   // sequencer 2: S100-S199 等待到位 / S100-S199 CheckLineMode
   STEP ProcessStart:   // S100, max time T#10S, warning time T#7S
      // 自动等待开始运行
              R    #ioPM_Inface.InitialRun
              R    #ioPM_Inface.ProcessComplete
              R    #ioPM_Inface.ProcessStart
              S    #ioPM_Inface.InitialOK
              S    #ioPM_Inface.WaitRunning
          S1  N    #ioPM_Inface.ProcessResult:=0
   END_STEP
   TRANSITION Trans200 FROM ProcessStart TO MotorRun   // T100
      := TRUE;
   END_TRANSITION
   STEP "Process Finish_1":   // S237, max time T#10S, warning time T#7S
   END_STEP
   TRANSITION Trans250 FROM "Process Finish_1" TO "CheckMachine Mode_1"   // T249, jump
      := TRUE;
   END_TRANSITION
   STEP StopProcess:   // S27, max time T#10S, warning time T#7S
   END_STEP
   TRANSITION Trans34 FROM StopProcess TO (UnloadStoper_1, UnloadStoper_2, UnloadStoper_3, "CheckMachine Mode_1", "CheckMachine Mode_2", "CheckMachine Mode_3", "CheckMachine Mode_4")   // T33
      := TRUE;
   END_TRANSITION
   STEP MotorRun:   // S34, max time T#10S, warning time T#7S
              S    "MotorControl".Dev[11].Auto.Start
              R    "MotorControl".Dev[11].Auto.CCWStart
              S    "MotorControl".Dev[12].Auto.Start
              R    "MotorControl".Dev[12].Auto.CCWStart
   END_STEP
   TRANSITION Trans39 FROM MotorRun TO StopProcess   // T38
      := TRUE;
   END_TRANSITION
   STEP LoadingStop_4:   // S30, max time T#10S, warning time T#7S
   END_STEP
   TRANSITION Trans122 FROM LoadingStop_4 TO CheckPalletExist_3   // T122
      := TRUE;
   END_TRANSITION
   STEP LoadingStop_2:   // S28, max time T#10S, warning time T#7S
   END_STEP
   TRANSITION Trans120 FROM LoadingStop_2 TO CheckPalletExist_1   // T120
      := TRUE;
   END_TRANSITION
   STEP "CheckMachine Mode_3":   // S156, max time T#10S, warning time T#7S
   END_STEP
   TRANSITION Trans166 FROM "CheckMachine Mode_3" TO LoadingStop_3   // T166
      := NOT "AutoProcessControl".Global.H.EmptyPallet;
   END_TRANSITION
   STEP LoadingStop_3:   // S29, max time T#10S, warning time T#7S
   END_STEP
   TRANSITION Trans121 FROM LoadingStop_3 TO CheckPalletExist_2   // T121
      := TRUE;
   END_TRANSITION
   STEP CheckPalletExist:   // S31, max time T#10S, warning time T#7S
              R    "MotorControl".Dev[11].Auto.CCWStart
   END_STEP
   TRANSITION Trans35 FROM CheckPalletExist TO WaitLineMotorReady   // T34
      := "iH-shaftLoadingDetection1" AND (#CheckPalletExist.T > t#1000MS) AND NOT "AutoProcessControl".Robot_1.ClearPart;
   END_TRANSITION
   STEP AriveTimeDelay_1:   // S119, max time T#10S, warning time T#7S
   END_STEP
   TRANSITION Trans119 FROM AriveTimeDelay_1 TO StoperReset_1   // T119
      := #AriveTimeDelay_1.T > t#500MS;
   END_TRANSITION
   STEP WaitLineMotorReady:   // S35, max time T#10S, warning time T#7S
   END_STEP
   TRANSITION Trans40 FROM WaitLineMotorReady TO WaitPalletRequestRelease   // T39
      := "MotorControl".Dev[11].OutControl.o_Ready;
   END_TRANSITION
   STEP WaitPalletRequestRelease:   // S36, max time T#10S, warning time T#7S
   END_STEP
   TRANSITION Trans41 FROM WaitPalletRequestRelease TO StoperRelease_1   // T40
      := "AutoProcessControl".Global.H.LoadStopRequestPallet_1;
   END_TRANSITION
   TRANSITION Trans207 FROM WaitPalletRequestRelease TO "CheckMachine Mode_1"   // T207, jump
      := "AutoProcessControl".Global.H.EmptyPallet;
   END_TRANSITION
   STEP LoadingStop_1:   // S142, max time T#10S, warning time T#7S
   END_STEP
   TRANSITION Trans776 FROM LoadingStop_1 TO CheckPalletExist   // T141
      := TRUE;
   END_TRANSITION
   STEP WaitPalletArrveNextPos:   // S37, max time T#10S, warning time T#7S
              S    "MotorControl".Dev[11].Auto.Start
              R    "MotorControl".Dev[11].Auto.CCWStart
   END_STEP
   TRANSITION Trans42 FROM WaitPalletArrveNextPos TO AriveTimeDelay_1   // T41
      := "iH-shaftLoadingDetection2" OR "AutoProcessControl".Global.H.EmptyPallet;
   END_TRANSITION
   STEP "Process Finish_2":   // S238, max time T#10S, warning time T#7S
   END_STEP
   TRANSITION Trans251 FROM "Process Finish_2" TO "CheckMachine Mode_2"   // T250, jump
      := TRUE;
   END_TRANSITION
   STEP StoperReset_1:   // S117, max time T#10S, warning time T#7S
              S    "ST10Cylinder".Cy[23].Inout.AutoGoHome
              R    "ST10Cylinder".Cy[23].Inout.AutoGoWork
   END_STEP
   TRANSITION Trans766 FROM StoperReset_1 TO "Process Finish_1"   // T117
      := TRUE;
   END_TRANSITION
   STEP StoperRelease_1:   // S118, max time T#10S, warning time T#7S
              R    "ST10Cylinder".Cy[23].Inout.AutoGoHome
              S    "ST10Cylinder".Cy[23].Inout.AutoGoWork
   END_STEP
   TRANSITION Trans767 FROM StoperRelease_1 TO WaitPalletArrveNextPos   // T118
      := #StoperRelease_1.T > t#1000MS;
   END_TRANSITION
   STEP CheckPalletExist_1:   // S32, max time T#10S, warning time T#7S
   END_STEP
   TRANSITION Trans36 FROM CheckPalletExist_1 TO WaitLineMotorReady_1   // T35
      := "iH-shaftLoadingDetection2" AND (#CheckPalletExist_1.T > t#1000MS);
   END_TRANSITION
   TRANSITION Trans126 FROM CheckPalletExist_1 TO WaitPalletArive   // T126
      := NOT "iH-shaftLoadingDetection2" AND (#CheckPalletExist_1.T > t#1000MS);
   END_TRANSITION
   STEP AriveTimeDelay_2:   // S120, max time T#10S, warning time T#7S
   END_STEP
   TRANSITION Trans123 FROM AriveTimeDelay_2 TO StoperReset_2   // T123
      := #AriveTimeDelay_2.T > t#500MS;
   END_TRANSITION
   STEP WaitLineMotorReady_1:   // S38, max time T#10S, warning time T#7S
   END_STEP
   TRANSITION Trans44 FROM WaitLineMotorReady_1 TO WaitPalletRequestRelease_1   // T43
      := "MotorControl".Dev[11].OutControl.o_Ready;
   END_TRANSITION
   STEP WaitPalletRequestRelease_1:   // S39, max time T#10S, warning time T#7S
   END_STEP
   TRANSITION Trans45 FROM WaitPalletRequestRelease_1 TO StoperRelease_2   // T44
      := "AutoProcessControl".Global.H.LoadStopRequestPallet_2;
   END_TRANSITION
   TRANSITION Trans206 FROM WaitPalletRequestRelease_1 TO "CheckMachine Mode_2"   // T206, jump
      := "AutoProcessControl".Global.H.EmptyPallet;
   END_TRANSITION
   STEP WaitPalletArrveNextPos_1:   // S40, max time T#10S, warning time T#7S
              S    "MotorControl".Dev[11].Auto.Start
              R    "MotorControl".Dev[11].Auto.CCWStart
   END_STEP
   TRANSITION Trans43 FROM WaitPalletArrveNextPos_1 TO AriveTimeDelay_2   // T42
      := "iH-shaftLoadingDetection3" OR "AutoProcessControl".Global.H.EmptyPallet;
   END_TRANSITION
   STEP StoperReset_2:   // S121, max time T#10S, warning time T#7S
              S    "ST10Cylinder".Cy[24].Inout.AutoGoHome
              R    "ST10Cylinder".Cy[24].Inout.AutoGoWork
   END_STEP
   TRANSITION Trans768 FROM StoperReset_2 TO "Process Finish_2"   // T124
      := TRUE;
   END_TRANSITION
   STEP StoperRelease_2:   // S122, max time T#10S, warning time T#7S
              R    "ST10Cylinder".Cy[24].Inout.AutoGoHome
              S    "ST10Cylinder".Cy[24].Inout.AutoGoWork
   END_STEP
   TRANSITION Trans769 FROM StoperRelease_2 TO WaitPalletArrveNextPos_1   // T125
      := #StoperRelease_2.T > t#1000MS;
   END_TRANSITION
   STEP WaitPalletArive:   // S123, max time T#10S, warning time T#7S
              N    "AutoProcessControl".Global.H.LoadStopRequestPallet_1
   END_STEP
   TRANSITION Trans127 FROM WaitPalletArive TO TimeDelay   // T127
      := "iH-shaftLoadingDetection2" OR "AutoProcessControl".Global.H.EmptyPallet;
   END_TRANSITION
   STEP TimeDelay:   // S124, max time T#10S, warning time T#7S
   END_STEP
   TRANSITION Trans128 FROM TimeDelay TO "CheckMachine Mode_2"   // T128, jump
      := #TimeDelay.T > t#500MS;
   END_TRANSITION
   STEP "Process Finish_3":   // S239, max time T#10S, warning time T#7S
   END_STEP
   TRANSITION Trans252 FROM "Process Finish_3" TO "CheckMachine Mode_3"   // T251, jump
      := TRUE;
   END_TRANSITION
   STEP CheckPalletExist_2:   // S41, max time T#10S, warning time T#7S
   END_STEP
   TRANSITION Trans37 FROM CheckPalletExist_2 TO WaitLineMotorReady_2   // T36
      := "iH-shaftLoadingDetection3" AND (#CheckPalletExist_2.T > t#1000MS);
   END_TRANSITION
   TRANSITION Trans129 FROM CheckPalletExist_2 TO WaitPalletArive_1   // T132
      := NOT "iH-shaftLoadingDetection3" AND (#CheckPalletExist_2.T > t#1000MS);
   END_TRANSITION
   STEP AriveTimeDelay_3:   // S125, max time T#10S, warning time T#7S
   END_STEP
   TRANSITION Trans124 FROM AriveTimeDelay_3 TO StoperReset_3   // T129
      := #AriveTimeDelay_3.T > t#500MS;
   END_TRANSITION
   STEP WaitLineMotorReady_2:   // S42, max time T#10S, warning time T#7S
   END_STEP
   TRANSITION Trans47 FROM WaitLineMotorReady_2 TO WaitPalletRequestRelease_2   // T46
      := "MotorControl".Dev[11].OutControl.o_Ready;
   END_TRANSITION
   STEP WaitPalletRequestRelease_2:   // S43, max time T#10S, warning time T#7S
   END_STEP
   TRANSITION Trans48 FROM WaitPalletRequestRelease_2 TO StoperRelease_3   // T47
      := "AutoProcessControl".Global.H.LoadStopRequestPallet_3;
   END_TRANSITION
   TRANSITION Trans205 FROM WaitPalletRequestRelease_2 TO "CheckMachine Mode_3"   // T205, jump
      := "AutoProcessControl".Global.H.EmptyPallet;
   END_TRANSITION
   STEP WaitPalletArrveNextPos_2:   // S44, max time T#10S, warning time T#7S
              S    "MotorControl".Dev[11].Auto.Start
              R    "MotorControl".Dev[11].Auto.CCWStart
   END_STEP
   TRANSITION Trans46 FROM WaitPalletArrveNextPos_2 TO AriveTimeDelay_3   // T45
      := "iH-shaftLoadingDetection4" OR "AutoProcessControl".Global.H.EmptyPallet;
   END_TRANSITION
   STEP StoperReset_3:   // S126, max time T#10S, warning time T#7S
              S    "ST10Cylinder".Cy[25].Inout.AutoGoHome
              R    "ST10Cylinder".Cy[25].Inout.AutoGoWork
   END_STEP
   TRANSITION Trans770 FROM StoperReset_3 TO "Process Finish_3"   // T130
      := TRUE;
   END_TRANSITION
   STEP StoperRelease_3:   // S127, max time T#10S, warning time T#7S
              R    "ST10Cylinder".Cy[25].Inout.AutoGoHome
              S    "ST10Cylinder".Cy[25].Inout.AutoGoWork
   END_STEP
   TRANSITION Trans771 FROM StoperRelease_3 TO WaitPalletArrveNextPos_2   // T131
      := #StoperRelease_3.T > t#1000MS;
   END_TRANSITION
   STEP WaitPalletArive_1:   // S128, max time T#10S, warning time T#7S
              N    "AutoProcessControl".Global.H.LoadStopRequestPallet_2
   END_STEP
   TRANSITION Trans130 FROM WaitPalletArive_1 TO TimeDelay_1   // T133
      := "iH-shaftLoadingDetection3" OR "AutoProcessControl".Global.H.EmptyPallet;
   END_TRANSITION
   STEP TimeDelay_1:   // S129, max time T#10S, warning time T#7S
   END_STEP
   TRANSITION Trans131 FROM TimeDelay_1 TO "CheckMachine Mode_3"   // T134, jump
      := #TimeDelay_1.T > t#500MS;
   END_TRANSITION
   STEP UnloadStoper_1:   // S201, max time T#10S, warning time T#7S
   END_STEP
   TRANSITION Trans125 FROM UnloadStoper_1 TO CheckPalletExist_4   // T135
      := TRUE;
   END_TRANSITION
   STEP "Process Finish_4":   // S240, max time T#10S, warning time T#7S
   END_STEP
   TRANSITION Trans253 FROM "Process Finish_4" TO "CheckMachine Mode_4"   // T252, jump
      := TRUE;
   END_TRANSITION
   STEP CheckPalletExist_3:   // S45, max time T#10S, warning time T#7S
   END_STEP
   TRANSITION Trans50 FROM CheckPalletExist_3 TO WaitLineMotorReady_3   // T49
      := "iH-shaftLoadingDetection4" AND (#CheckPalletExist_3.T > t#1000MS);
   END_TRANSITION
   TRANSITION Trans133 FROM CheckPalletExist_3 TO WaitPalletArive_2   // T139
      := NOT "iH-shaftLoadingDetection4" AND (#CheckPalletExist_3.T > t#1000MS);
   END_TRANSITION
   STEP AriveTimeDelay_4:   // S130, max time T#10S, warning time T#7S
   END_STEP
   TRANSITION Trans132 FROM AriveTimeDelay_4 TO StoperReset_4   // T136
      := #AriveTimeDelay_4.T > t#500MS;
   END_TRANSITION
   STEP WaitLineMotorReady_3:   // S46, max time T#10S, warning time T#7S
   END_STEP
   TRANSITION Trans51 FROM WaitLineMotorReady_3 TO WaitPalletRequestRelease_3   // T50
      := "MotorControl".Dev[11].OutControl.o_Ready;
   END_TRANSITION
   STEP WaitPalletRequestRelease_3:   // S47, max time T#10S, warning time T#7S
   END_STEP
   TRANSITION Trans52 FROM WaitPalletRequestRelease_3 TO StoperRelease_4   // T51
      := "AutoProcessControl".Global.H.LoadStopRequestPallet_4;
   END_TRANSITION
   TRANSITION Trans204 FROM WaitPalletRequestRelease_3 TO "CheckMachine Mode_4"   // T204, jump
      := "AutoProcessControl".Global.H.EmptyPallet;
   END_TRANSITION
   STEP WaitPalletArrveNextPos_3:   // S48, max time T#10S, warning time T#7S
              S    "MotorControl".Dev[11].Auto.Start
              R    "MotorControl".Dev[11].Auto.CCWStart
              R    "MotorControl".Dev[1].Auto.CCWStart
              S    "MotorControl".Dev[1].Auto.Start
   END_STEP
   TRANSITION Trans49 FROM WaitPalletArrveNextPos_3 TO AriveTimeDelay_4   // T48
      := ("iH-shaftLiftingPalletDischarge" AND NOT "iH-shaftMiddleDetection") OR "AutoProcessControl".Global.H.EmptyPallet;
   END_TRANSITION
   STEP StoperReset_4:   // S131, max time T#10S, warning time T#7S
              S    "ST10Cylinder".Cy[26].Inout.AutoGoHome
              R    "ST10Cylinder".Cy[26].Inout.AutoGoWork
   END_STEP
   TRANSITION Trans772 FROM StoperReset_4 TO "Process Finish_4"   // T137
      := TRUE;
   END_TRANSITION
   STEP StoperRelease_4:   // S133, max time T#10S, warning time T#7S
              R    "ST10Cylinder".Cy[26].Inout.AutoGoHome
              S    "ST10Cylinder".Cy[26].Inout.AutoGoWork
   END_STEP
   TRANSITION Trans773 FROM StoperRelease_4 TO WaitPalletArrveNextPos_3   // T138
      := #StoperRelease_4.T > t#1000MS;
   END_TRANSITION
   STEP WaitPalletArive_2:   // S134, max time T#10S, warning time T#7S
              N    "AutoProcessControl".Global.H.LoadStopRequestPallet_3
   END_STEP
   TRANSITION Trans134 FROM WaitPalletArive_2 TO TimeDelay_2   // T140
      := "iH-shaftLoadingDetection4" OR "AutoProcessControl".Global.H.EmptyPallet;
   END_TRANSITION
   STEP TimeDelay_2:   // S135, max time T#10S, warning time T#7S
   END_STEP
   TRANSITION Trans135 FROM TimeDelay_2 TO "CheckMachine Mode_4"   // T144, jump
      := #TimeDelay_2.T > t#500MS;
   END_TRANSITION
   STEP UnloadStoper_2:   // S202, max time T#10S, warning time T#7S
   END_STEP
   TRANSITION Trans202 FROM UnloadStoper_2 TO CheckPalletExist_5   // T202
      := TRUE;
   END_TRANSITION
   STEP UnloadStoper_3:   // S203, max time T#10S, warning time T#7S
   END_STEP
   TRANSITION Trans203 FROM UnloadStoper_3 TO CheckPalletExist_6   // T203
      := TRUE;
   END_TRANSITION
   STEP "Process Finish_6":   // S242, max time T#10S, warning time T#7S
   END_STEP
   TRANSITION Trans255 FROM "Process Finish_6" TO UnloadStoper_2   // T254, jump
      := TRUE;
   END_TRANSITION
   STEP "Process Finish_5":   // S241, max time T#10S, warning time T#7S
   END_STEP
   TRANSITION Trans254 FROM "Process Finish_5" TO UnloadStoper_1   // T253, jump
      := TRUE;
   END_TRANSITION
   STEP CheckPalletExist_4:   // S49, max time T#10S, warning time T#7S
   END_STEP
   TRANSITION Trans54 FROM CheckPalletExist_4 TO WaitLineMotorReady_4   // T53
      := "iH-shaftTakeDetection1" AND (#CheckPalletExist_4.T > t#1000MS);
   END_TRANSITION
   TRANSITION Trans137 FROM CheckPalletExist_4 TO WaitPalletArive_3   // T148
      := NOT "iH-shaftTakeDetection1" AND (#CheckPalletExist_4.T > t#1000MS);
   END_TRANSITION
   STEP AriveTimeDelay_5:   // S136, max time T#10S, warning time T#7S
   END_STEP
   TRANSITION Trans136 FROM AriveTimeDelay_5 TO StoperReset_5   // T145
      := #AriveTimeDelay_5.T > t#500MS;
   END_TRANSITION
   STEP WaitLineMotorReady_4:   // S50, max time T#10S, warning time T#7S
   END_STEP
   TRANSITION Trans55 FROM WaitLineMotorReady_4 TO WaitPalletRequestRelease_4   // T54
      := "MotorControl".Dev[12].OutControl.o_Ready;
   END_TRANSITION
   STEP WaitPalletRequestRelease_4:   // S51, max time T#10S, warning time T#7S
   END_STEP
   TRANSITION Trans56 FROM WaitPalletRequestRelease_4 TO StoperRelease_5   // T55
      := "AutoProcessControl".Global.H.EmptyStopRequestPallet_2;
   END_TRANSITION
   STEP WaitPalletArrveNextPos_4:   // S52, max time T#10S, warning time T#7S
              S    "MotorControl".Dev[12].Auto.Start
              R    "MotorControl".Dev[12].Auto.CCWStart
   END_STEP
   TRANSITION Trans53 FROM WaitPalletArrveNextPos_4 TO AriveTimeDelay_5   // T52
      := "iH-shaftTakeDetection2";
   END_TRANSITION
   STEP StoperReset_5:   // S137, max time T#10S, warning time T#7S
              S    "ST10Cylinder".Cy[27].Inout.AutoGoHome
              R    "ST10Cylinder".Cy[27].Inout.AutoGoWork
   END_STEP
   TRANSITION Trans774 FROM StoperReset_5 TO "Process Finish_5"   // T146
      := TRUE;
   END_TRANSITION
   STEP StoperRelease_5:   // S138, max time T#10S, warning time T#7S
              R    "ST10Cylinder".Cy[27].Inout.AutoGoHome
              S    "ST10Cylinder".Cy[27].Inout.AutoGoWork
   END_STEP
   TRANSITION Trans775 FROM StoperRelease_5 TO WaitPalletArrveNextPos_4   // T147
      := #StoperRelease_5.T > t#1000MS;
   END_TRANSITION
   STEP WaitPalletArive_3:   // S139, max time T#10S, warning time T#7S
      interlock C := "ST10Cylinder".Cy[27].Inout.AutoGoHome AND NOT "ST10Cylinder".Cy[27].Inout.AutoGoWork;
      (C)     N    "AutoProcessControl".Global.H.EmptyStopRequestPallet_1
   END_STEP
   TRANSITION Trans138 FROM WaitPalletArive_3 TO TimeDelay_3   // T149
      := "iH-shaftTakeDetection1";
   END_TRANSITION
   STEP TimeDelay_3:   // S140, max time T#10S, warning time T#7S
   END_STEP
   TRANSITION Trans139 FROM TimeDelay_3 TO UnloadStoper_1   // T150, jump
      := #TimeDelay_3.T > t#500MS;
   END_TRANSITION
   STEP CheckPalletExist_5:   // S53, max time T#10S, warning time T#7S
   END_STEP
   TRANSITION Trans58 FROM CheckPalletExist_5 TO WaitLineMotorReady_5   // T57
      := "iH-shaftTakeDetection2" AND (#CheckPalletExist_5.T > t#1000MS);
   END_TRANSITION
   TRANSITION Trans141 FROM CheckPalletExist_5 TO WaitPalletArive_4   // T154
      := NOT "iH-shaftTakeDetection2" AND (#CheckPalletExist_5.T > t#1000MS);
   END_TRANSITION
   STEP AriveTimeDelay_6:   // S141, max time T#10S, warning time T#7S
   END_STEP
   TRANSITION Trans140 FROM AriveTimeDelay_6 TO StoperReset_6   // T151
      := #AriveTimeDelay_6.T > t#500MS;
   END_TRANSITION
   STEP WaitLineMotorReady_5:   // S54, max time T#10S, warning time T#7S
   END_STEP
   TRANSITION Trans59 FROM WaitLineMotorReady_5 TO WaitPalletRequestRelease_5   // T58
      := "MotorControl".Dev[12].OutControl.o_Ready;
   END_TRANSITION
   STEP WaitPalletRequestRelease_5:   // S55, max time T#10S, warning time T#7S
   END_STEP
   TRANSITION Trans60 FROM WaitPalletRequestRelease_5 TO StoperRelease_6   // T59
      := "AutoProcessControl".Global.H.EmptyStopRequestPallet_3;
   END_TRANSITION
   STEP WaitPalletArrveNextPos_5:   // S56, max time T#10S, warning time T#7S
              S    "MotorControl".Dev[12].Auto.Start
              R    "MotorControl".Dev[12].Auto.CCWStart
   END_STEP
   TRANSITION Trans57 FROM WaitPalletArrveNextPos_5 TO AriveTimeDelay_6   // T56
      := "iH-shaftTakeDetection3";
   END_TRANSITION
   STEP StoperReset_6:   // S144, max time T#10S, warning time T#7S
              S    "ST10Cylinder".Cy[28].Inout.AutoGoHome
              R    "ST10Cylinder".Cy[28].Inout.AutoGoWork
   END_STEP
   TRANSITION Trans777 FROM StoperReset_6 TO "Process Finish_6"   // T152
      := TRUE;
   END_TRANSITION
   STEP StoperRelease_6:   // S145, max time T#10S, warning time T#7S
              R    "ST10Cylinder".Cy[28].Inout.AutoGoHome
              S    "ST10Cylinder".Cy[28].Inout.AutoGoWork
   END_STEP
   TRANSITION Trans778 FROM StoperRelease_6 TO WaitPalletArrveNextPos_5   // T153
      := #StoperRelease_6.T > t#1000MS;
   END_TRANSITION
   STEP WaitPalletArive_4:   // S146, max time T#10S, warning time T#7S
              N    "AutoProcessControl".Global.H.EmptyStopRequestPallet_2
   END_STEP
   TRANSITION Trans144 FROM WaitPalletArive_4 TO TimeDelay_4   // T155
      := "iH-shaftTakeDetection2";
   END_TRANSITION
   STEP TimeDelay_4:   // S147, max time T#10S, warning time T#7S
   END_STEP
   TRANSITION Trans146 FROM TimeDelay_4 TO UnloadStoper_2   // T156, jump
      := #TimeDelay_4.T > t#500MS;
   END_TRANSITION
   STEP "CheckMachine Mode_1":   // S154, max time T#10S, warning time T#7S
   END_STEP
   TRANSITION Trans164 FROM "CheckMachine Mode_1" TO LoadingStop_1   // T164
      := NOT "AutoProcessControl".Global.H.EmptyPallet;
   END_TRANSITION
   STEP "Process Finish_7":   // S243, max time T#10S, warning time T#7S
   END_STEP
   TRANSITION Trans256 FROM "Process Finish_7" TO UnloadStoper_3   // T255, jump
      := TRUE;
   END_TRANSITION
   STEP CheckPalletExist_6:   // S57, max time T#10S, warning time T#7S
   END_STEP
   TRANSITION Trans62 FROM CheckPalletExist_6 TO WaitLineMotorReady_6   // T61
      := "iH-shaftTakeDetection3" AND (#CheckPalletExist_6.T > t#1000MS);
   END_TRANSITION
   TRANSITION Trans148 FROM CheckPalletExist_6 TO WaitPalletArive_5   // T160
      := NOT "iH-shaftTakeDetection3" AND (#CheckPalletExist_6.T > t#1000MS);
   END_TRANSITION
   STEP AriveTimeDelay_7:   // S148, max time T#10S, warning time T#7S
   END_STEP
   TRANSITION Trans147 FROM AriveTimeDelay_7 TO StoperReset_7   // T157
      := #AriveTimeDelay_7.T > t#500MS;
   END_TRANSITION
   STEP WaitLineMotorReady_6:   // S58, max time T#10S, warning time T#7S
   END_STEP
   TRANSITION Trans63 FROM WaitLineMotorReady_6 TO WaitPalletRequestRelease_6   // T62
      := "MotorControl".Dev[12].OutControl.o_Ready;
   END_TRANSITION
   STEP WaitPalletRequestRelease_6:   // S59, max time T#10S, warning time T#7S
   END_STEP
   TRANSITION Trans64 FROM WaitPalletRequestRelease_6 TO StoperRelease_7   // T63
      := NOT "iH-shaftTakeShaftDetection";
   END_TRANSITION
   STEP WaitPalletArrveNextPos_6:   // S60, max time T#10S, warning time T#7S
              S    "MotorControl".Dev[12].Auto.Start
              R    "MotorControl".Dev[12].Auto.CCWStart
   END_STEP
   TRANSITION Trans61 FROM WaitPalletArrveNextPos_6 TO AriveTimeDelay_7   // T60
      := "iH-shaftTakeShaftDetection";
   END_TRANSITION
   STEP StoperReset_7:   // S149, max time T#10S, warning time T#7S
              S    "ST10Cylinder".Cy[29].Inout.AutoGoHome
              R    "ST10Cylinder".Cy[29].Inout.AutoGoWork
   END_STEP
   TRANSITION Trans779 FROM StoperReset_7 TO "Process Finish_7"   // T158
      := TRUE;
   END_TRANSITION
   STEP StoperRelease_7:   // S150, max time T#10S, warning time T#7S
              R    "ST10Cylinder".Cy[29].Inout.AutoGoHome
              S    "ST10Cylinder".Cy[29].Inout.AutoGoWork
   END_STEP
   TRANSITION Trans780 FROM StoperRelease_7 TO WaitPalletArrveNextPos_6   // T159
      := #StoperRelease_7.T > t#1000MS;
   END_TRANSITION
   STEP WaitPalletArive_5:   // S151, max time T#10S, warning time T#7S
              N    "AutoProcessControl".Global.H.EmptyStopRequestPallet_3
   END_STEP
   TRANSITION Trans149 FROM WaitPalletArive_5 TO TimeDelay_5   // T161
      := "iH-shaftTakeDetection3";
   END_TRANSITION
   STEP TimeDelay_5:   // S152, max time T#10S, warning time T#7S
   END_STEP
   TRANSITION Trans150 FROM TimeDelay_5 TO UnloadStoper_3   // T162, jump
      := #TimeDelay_5.T > t#500MS;
   END_TRANSITION
   STEP "CheckMachine Mode_2":   // S155, max time T#10S, warning time T#7S
   END_STEP
   TRANSITION Trans165 FROM "CheckMachine Mode_2" TO LoadingStop_2   // T165
      := NOT "AutoProcessControl".Global.H.EmptyPallet;
   END_TRANSITION
   STEP "CheckMachine Mode_4":   // S157, max time T#10S, warning time T#7S
   END_STEP
   TRANSITION Trans167 FROM "CheckMachine Mode_4" TO LoadingStop_4   // T167
      := NOT "AutoProcessControl".Global.H.EmptyPallet;
   END_TRANSITION

   // sequencer 3: Empty Process
   INITIAL_STEP CheckMachineMode:   // S200, max time T#10S, warning time T#7S
   END_STEP
   TRANSITION Trans145 FROM CheckMachineMode TO WaitAllStoperReset   // T200
      := "AutoProcessControl".Global.H.EmptyPallet;
   END_TRANSITION
   STEP Step153:   // S153, max time T#10S, warning time T#7S
   END_STEP
   TRANSITION Trans163 FROM Step153 TO "CheckMachine Mode_6"   // T163, jump
      := TRUE;
   END_TRANSITION
   STEP "Process Finish_8":   // S244, max time T#10S, warning time T#7S
   END_STEP
   TRANSITION Trans257 FROM "Process Finish_8" TO Step153   // T256
      := TRUE;
   END_TRANSITION
   STEP LoadStop_14:   // S61, max time T#10S, warning time T#7S
   END_STEP
   TRANSITION Trans154 FROM LoadStop_14 TO CheckPalletExist_10   // T175
      := #LoadStop_14.T > t#2S;
   END_TRANSITION
   STEP LoadStop_12:   // S62, max time T#10S, warning time T#7S
   END_STEP
   TRANSITION Trans152 FROM LoadStop_12 TO CheckPalletExist_8   // T169
      := #LoadStop_12.T > t#2S;
   END_TRANSITION
   STEP "CheckMachine Mode_5":   // S158, max time T#10S, warning time T#7S
   END_STEP
   TRANSITION Trans175 FROM "CheckMachine Mode_5" TO LoadStop_13   // T196
      := "AutoProcessControl".Global.H.EmptyPallet;
   END_TRANSITION
   STEP LoadStop_13:   // S63, max time T#10S, warning time T#7S
   END_STEP
   TRANSITION Trans153 FROM LoadStop_13 TO CheckPalletExist_9   // T170
      := #LoadStop_13.T > t#2S;
   END_TRANSITION
   STEP CheckPalletExist_7:   // S64, max time T#10S, warning time T#7S
   END_STEP
   TRANSITION Trans66 FROM CheckPalletExist_7 TO WaitLineMotorReady_7   // T65
      := "H-shaftPalletEmptyCheck1" AND (#CheckPalletExist_7.T > t#1000MS);
   END_TRANSITION
   TRANSITION Trans33 FROM CheckPalletExist_7 TO WaitPalletArive_9   // T32
      := NOT "H-shaftPalletEmptyCheck1" AND (#CheckPalletExist_7.T > t#1000MS);
   END_TRANSITION
   STEP AriveTimeDelay_8:   // S159, max time T#10S, warning time T#7S
   END_STEP
   TRANSITION Trans151 FROM AriveTimeDelay_8 TO StoperReset_8   // T168
      := #AriveTimeDelay_8.T > t#500MS;
   END_TRANSITION
   STEP WaitLineMotorReady_7:   // S65, max time T#10S, warning time T#7S
   END_STEP
   TRANSITION Trans67 FROM WaitLineMotorReady_7 TO WaitPalletRequestRelease_7   // T66
      := "MotorControl".Dev[11].OutControl.o_Ready;
   END_TRANSITION
   STEP WaitPalletRequestRelease_7:   // S66, max time T#10S, warning time T#7S
   END_STEP
   TRANSITION Trans68 FROM WaitPalletRequestRelease_7 TO StoperRelease_8   // T67
      := NOT "iH-shaftTakeGateDetection";
   END_TRANSITION
   STEP LoadStop_11:   // S160, max time T#10S, warning time T#7S
   END_STEP
   TRANSITION Trans781 FROM LoadStop_11 TO CheckPalletExist_7   // T172
      := #LoadStop_11.T > t#2S;
   END_TRANSITION
   STEP WaitPalletArrveNextPos_7:   // S67, max time T#10S, warning time T#7S
   END_STEP
   TRANSITION Trans65 FROM WaitPalletArrveNextPos_7 TO AriveTimeDelay_8   // T64
      := "iH-shaftTakeGateDetection";
   END_TRANSITION
   STEP "Process Finish_9":   // S245, max time T#10S, warning time T#7S
   END_STEP
   TRANSITION Trans258 FROM "Process Finish_9" TO "CheckMachine Mode_7"   // T257, jump
      := TRUE;
   END_TRANSITION
   STEP StoperReset_8:   // S161, max time T#10S, warning time T#7S
              S    "ST10Cylinder".Cy[23].Inout.AutoGoHome
              R    "ST10Cylinder".Cy[23].Inout.AutoGoWork
   END_STEP
   TRANSITION Trans782 FROM StoperReset_8 TO "Process Finish_8"   // T173
      := TRUE;
   END_TRANSITION
   STEP StoperRelease_8:   // S162, max time T#10S, warning time T#7S
              R    "ST10Cylinder".Cy[23].Inout.AutoGoHome
              S    "ST10Cylinder".Cy[23].Inout.AutoGoWork
   END_STEP
   TRANSITION Trans783 FROM StoperRelease_8 TO WaitPalletArrveNextPos_7   // T174
      := #StoperRelease_8.T > t#1000MS;
   END_TRANSITION
   STEP CheckPalletExist_8:   // S68, max time T#10S, warning time T#7S
   END_STEP
   TRANSITION Trans70 FROM CheckPalletExist_8 TO WaitLineMotorReady_8   // T69
      := "H-shaftPalletEmptyCheck2" AND (#CheckPalletExist_8.T > t#1000MS);
   END_TRANSITION
   TRANSITION Trans156 FROM CheckPalletExist_8 TO WaitPalletArive_6   // T179
      := NOT "H-shaftPalletEmptyCheck2" AND (#CheckPalletExist_8.T > t#1000MS);
   END_TRANSITION
   STEP AriveTimeDelay_9:   // S163, max time T#10S, warning time T#7S
   END_STEP
   TRANSITION Trans155 FROM AriveTimeDelay_9 TO StoperReset_9   // T176
      := #AriveTimeDelay_9.T > t#500MS;
   END_TRANSITION
   STEP WaitLineMotorReady_8:   // S69, max time T#10S, warning time T#7S
   END_STEP
   TRANSITION Trans71 FROM WaitLineMotorReady_8 TO WaitPalletRequestRelease_8   // T70
      := "MotorControl".Dev[11].OutControl.o_Ready;
   END_TRANSITION
   STEP WaitPalletRequestRelease_8:   // S70, max time T#10S, warning time T#7S
   END_STEP
   TRANSITION Trans72 FROM WaitPalletRequestRelease_8 TO StoperRelease_9   // T71
      := "AutoProcessControl".Global.H.LoadStopRequestPallet_2;
   END_TRANSITION
   STEP WaitPalletArrveNextPos_8:   // S71, max time T#10S, warning time T#7S
   END_STEP
   TRANSITION Trans69 FROM WaitPalletArrveNextPos_8 TO AriveTimeDelay_9   // T68
      := "H-shaftPalletEmptyCheck1";
   END_TRANSITION
   STEP StoperReset_9:   // S164, max time T#10S, warning time T#7S
              S    "ST10Cylinder".Cy[24].Inout.AutoGoHome
              R    "ST10Cylinder".Cy[24].Inout.AutoGoWork
   END_STEP
   TRANSITION Trans784 FROM StoperReset_9 TO "Process Finish_9"   // T177
      := TRUE;
   END_TRANSITION
   STEP StoperRelease_9:   // S165, max time T#10S, warning time T#7S
              R    "ST10Cylinder".Cy[24].Inout.AutoGoHome
              S    "ST10Cylinder".Cy[24].Inout.AutoGoWork
   END_STEP
   TRANSITION Trans785 FROM StoperRelease_9 TO WaitPalletArrveNextPos_8   // T178
      := #StoperRelease_9.T > t#1000MS;
   END_TRANSITION
   STEP WaitPalletArive_6:   // S166, max time T#10S, warning time T#7S
              N    "AutoProcessControl".Global.H.LoadStopRequestPallet_3
   END_STEP
   TRANSITION Trans157 FROM WaitPalletArive_6 TO TimeDelay_6   // T180
      := "H-shaftPalletEmptyCheck2" OR NOT "AutoProcessControl".Global.H.EmptyPallet;
   END_TRANSITION
   STEP TimeDelay_6:   // S167, max time T#10S, warning time T#7S
   END_STEP
   TRANSITION Trans158 FROM TimeDelay_6 TO "CheckMachine Mode_7"   // T181, jump
      := #TimeDelay_6.T > t#500MS;
   END_TRANSITION
   STEP "Process Finish_10":   // S246, max time T#10S, warning time T#7S
   END_STEP
   TRANSITION Trans259 FROM "Process Finish_10" TO "CheckMachine Mode_5"   // T258, jump
      := TRUE;
   END_TRANSITION
   STEP CheckPalletExist_9:   // S72, max time T#10S, warning time T#7S
   END_STEP
   TRANSITION Trans74 FROM CheckPalletExist_9 TO WaitLineMotorReady_9   // T73
      := "H-shaftPalletEmptyCheck3" AND (#CheckPalletExist_9.T > t#1000MS);
   END_TRANSITION
   TRANSITION Trans160 FROM CheckPalletExist_9 TO WaitPalletArive_7   // T185
      := NOT "H-shaftPalletEmptyCheck3" AND (#CheckPalletExist_9.T > t#1000MS);
   END_TRANSITION
   STEP AriveTimeDelay_10:   // S168, max time T#10S, warning time T#7S
   END_STEP
   TRANSITION Trans159 FROM AriveTimeDelay_10 TO StoperReset_10   // T182
      := #AriveTimeDelay_10.T > t#500MS;
   END_TRANSITION
   STEP WaitLineMotorReady_9:   // S73, max time T#10S, warning time T#7S
   END_STEP
   TRANSITION Trans75 FROM WaitLineMotorReady_9 TO WaitPalletRequestRelease_9   // T74
      := "MotorControl".Dev[11].OutControl.o_Ready;
   END_TRANSITION
   STEP WaitPalletRequestRelease_9:   // S74, max time T#10S, warning time T#7S
   END_STEP
   TRANSITION Trans76 FROM WaitPalletRequestRelease_9 TO StoperRelease_10   // T75
      := "AutoProcessControl".Global.H.LoadStopRequestPallet_3;
   END_TRANSITION
   STEP WaitPalletArrveNextPos_9:   // S75, max time T#10S, warning time T#7S
   END_STEP
   TRANSITION Trans73 FROM WaitPalletArrveNextPos_9 TO AriveTimeDelay_10   // T72
      := "H-shaftPalletEmptyCheck2";
   END_TRANSITION
   STEP StoperReset_10:   // S169, max time T#10S, warning time T#7S
              S    "ST10Cylinder".Cy[25].Inout.AutoGoHome
              R    "ST10Cylinder".Cy[25].Inout.AutoGoWork
   END_STEP
   TRANSITION Trans786 FROM StoperReset_10 TO "Process Finish_10"   // T183
      := TRUE;
   END_TRANSITION
   STEP StoperRelease_10:   // S170, max time T#10S, warning time T#7S
              R    "ST10Cylinder".Cy[25].Inout.AutoGoHome
              S    "ST10Cylinder".Cy[25].Inout.AutoGoWork
   END_STEP
   TRANSITION Trans787 FROM StoperRelease_10 TO WaitPalletArrveNextPos_9   // T184
      := #StoperRelease_10.T > t#1000MS;
   END_TRANSITION
   STEP WaitPalletArive_7:   // S171, max time T#10S, warning time T#7S
              N    "AutoProcessControl".Global.H.LoadStopRequestPallet_4
   END_STEP
   TRANSITION Trans161 FROM WaitPalletArive_7 TO TimeDelay_7   // T186
      := "H-shaftPalletEmptyCheck3" OR NOT "AutoProcessControl".Global.H.EmptyPallet;
   END_TRANSITION
   STEP TimeDelay_7:   // S172, max time T#10S, warning time T#7S
   END_STEP
   TRANSITION Trans162 FROM TimeDelay_7 TO "CheckMachine Mode_5"   // T187, jump
      := #TimeDelay_7.T > t#500MS;
   END_TRANSITION
   STEP "Process Finish_11":   // S247, max time T#10S, warning time T#7S
   END_STEP
   TRANSITION Trans260 FROM "Process Finish_11" TO "CheckMachine Mode_8"   // T259, jump
      := TRUE;
   END_TRANSITION
   STEP CheckPalletExist_10:   // S76, max time T#10S, warning time T#7S
   END_STEP
   TRANSITION Trans78 FROM CheckPalletExist_10 TO WaitLineMotorReady_10   // T77
      := "iH-shaftPalletEmptyCheck4" AND "iH-shaftMiddleDetection" AND (#CheckPalletExist_10.T > t#1000MS);
   END_TRANSITION
   TRANSITION Trans170 FROM CheckPalletExist_10 TO WaitPalletArive_8   // T191
      := NOT "iH-shaftPalletEmptyCheck4" AND (#CheckPalletExist_10.T > t#1000MS);
   END_TRANSITION
   STEP AriveTimeDelay_11:   // S173, max time T#10S, warning time T#7S
   END_STEP
   TRANSITION Trans169 FROM AriveTimeDelay_11 TO StoperReset_11   // T188
      := #AriveTimeDelay_11.T > t#500MS;
   END_TRANSITION
   STEP WaitLineMotorReady_10:   // S77, max time T#10S, warning time T#7S
   END_STEP
   TRANSITION Trans79 FROM WaitLineMotorReady_10 TO WaitPalletRequestRelease_10   // T78
      := "MotorControl".Dev[11].OutControl.o_Ready;
   END_TRANSITION
   STEP WaitPalletRequestRelease_10:   // S78, max time T#10S, warning time T#7S
   END_STEP
   TRANSITION Trans80 FROM WaitPalletRequestRelease_10 TO StoperRelease_11   // T79
      := "AutoProcessControl".Global.H.LoadStopRequestPallet_4;
   END_TRANSITION
   STEP WaitPalletArrveNextPos_10:   // S79, max time T#10S, warning time T#7S
   END_STEP
   TRANSITION Trans77 FROM WaitPalletArrveNextPos_10 TO AriveTimeDelay_11   // T76
      := "H-shaftPalletEmptyCheck3";
   END_TRANSITION
   STEP StoperReset_11:   // S174, max time T#10S, warning time T#7S
              S    "ST10Cylinder".Cy[26].Inout.AutoGoHome
              R    "ST10Cylinder".Cy[26].Inout.AutoGoWork
   END_STEP
   TRANSITION Trans788 FROM StoperReset_11 TO "Process Finish_11"   // T189
      := TRUE;
   END_TRANSITION
   STEP StoperRelease_11:   // S175, max time T#10S, warning time T#7S
              R    "ST10Cylinder".Cy[26].Inout.AutoGoHome
              S    "ST10Cylinder".Cy[26].Inout.AutoGoWork
   END_STEP
   TRANSITION Trans789 FROM StoperRelease_11 TO WaitPalletArrveNextPos_10   // T190
      := #StoperRelease_11.T > t#1000MS;
   END_TRANSITION
   STEP WaitPalletArive_8:   // S176, max time T#10S, warning time T#7S
   END_STEP
   TRANSITION Trans171 FROM WaitPalletArive_8 TO TimeDelay_8   // T192
      := ("iH-shaftPalletEmptyCheck4" AND "iH-shaftMiddleDetection") OR NOT "AutoProcessControl".Global.H.EmptyPallet;
   END_TRANSITION
   STEP TimeDelay_8:   // S177, max time T#10S, warning time T#7S
   END_STEP
   TRANSITION Trans172 FROM TimeDelay_8 TO "CheckMachine Mode_8"   // T193, jump
      := #TimeDelay_8.T > t#500MS;
   END_TRANSITION
   STEP "CheckMachine Mode_6":   // S178, max time T#10S, warning time T#7S
   END_STEP
   TRANSITION Trans173 FROM "CheckMachine Mode_6" TO LoadStop_11   // T194
      := "AutoProcessControl".Global.H.EmptyPallet;
   END_TRANSITION
   STEP "CheckMachine Mode_7":   // S179, max time T#10S, warning time T#7S
   END_STEP
   TRANSITION Trans174 FROM "CheckMachine Mode_7" TO LoadStop_12   // T195
      := "AutoProcessControl".Global.H.EmptyPallet;
   END_TRANSITION
   STEP "CheckMachine Mode_8":   // S180, max time T#10S, warning time T#7S
   END_STEP
   TRANSITION Trans168 FROM "CheckMachine Mode_8" TO LoadStop_14   // T171
      := "AutoProcessControl".Global.H.EmptyPallet;
   END_TRANSITION
   STEP WaitAllStoperReset:   // S181, max time T#10S, warning time T#7S
   END_STEP
   TRANSITION Trans197 FROM WaitAllStoperReset TO MotorRun_1   // T197
      := "ST10Cylinder".Cy[23].Inout.AutoGoHome AND NOT "ST10Cylinder".Cy[23].Inout.AutoGoWork AND "ST10Cylinder".Cy[24].Inout.AutoGoHome AND NOT "ST10Cylinder".Cy[24].Inout.AutoGoWork AND "ST10Cylinder".Cy[25].Inout.AutoGoHome AND NOT "ST10Cylinder".Cy[25].Inout.AutoGoWork AND "ST10Cylinder".Cy[26].Inout.AutoGoHome AND NOT "ST10Cylinder".Cy[26].Inout.AutoGoWork;
   END_TRANSITION
   STEP Step182:   // S182, max time T#10S, warning time T#7S
   END_STEP
   TRANSITION Trans198 FROM Step182 TO ("CheckMachine Mode_7", "CheckMachine Mode_5", "CheckMachine Mode_8", "CheckMachine Mode_6")   // T198
      := TRUE;
   END_TRANSITION
   STEP MotorRun_1:   // S80, max time T#10S, warning time T#7S
              R    "MotorControl".Dev[11].Auto.Start
              S    "MotorControl".Dev[11].Auto.CCWStart
              S    "MotorControl".Dev[12].Auto.Start
              R    "MotorControl".Dev[12].Auto.CCWStart
   END_STEP
   TRANSITION Trans81 FROM MotorRun_1 TO Step182   // T80
      := TRUE;
   END_TRANSITION
   STEP WaitPalletArive_9:   // S183, max time T#10S, warning time T#7S
              N    "AutoProcessControl".Global.H.LoadStopRequestPallet_2
   END_STEP
   TRANSITION Trans176 FROM WaitPalletArive_9 TO TimeDelay_9   // T199
      := "H-shaftPalletEmptyCheck1" OR NOT "AutoProcessControl".Global.H.EmptyPallet;
   END_TRANSITION
   STEP TimeDelay_9:   // S184, max time T#10S, warning time T#7S
   END_STEP
   TRANSITION Trans177 FROM TimeDelay_9 TO "CheckMachine Mode_6"   // T201, jump
      := #TimeDelay_9.T > t#500MS;
   END_TRANSITION

   // permanent post-instructions
   NETWORK 1
      #ioPM_Inface.StepNum := #RT_DATA.S_DISPLAY;
   NETWORK 2
      IF #iSysInface.Reset THEN #AlarmID := 0; END_IF;
   NETWORK 3
      #TON[10].TON(IN := #工件放行中, PT := T#0.5S);
      IF #TON[10].Q THEN #工件放行中 := FALSE; END_IF;
END_FUNCTION_BLOCK

FUNCTION_BLOCK "ST10_Flow26_JMagnetLoad&Unload"   // FB1096, GRAPH
// stored: AcknowledgeErrorsRequired false, AutoNumber false, GraphVersion 6.0, InitialValuesAcquisition false, SetENOAutomatically false
   // inherited from GRAPH_BASE
   VAR_INPUT
      iSysInface : "RCS_SysComInterface_V1";
   END_VAR
   VAR_IN_OUT
      ioPM_Inface : "RCS_PMInterface_V1";
      ioStatus : Int;
   END_VAR
   VAR
      sCtrlMode { S7_SetPoint := 'True'} : "SysFlowCtrlGraph";
      sUpdMES_Data : Bool;   // 更新MES数据
      工件放行中 : Bool;
      前站站号 { ExternalAccessible := 'False'; ExternalVisible := 'False'; ExternalWritable := 'False'} : UInt;
      本站站号 { ExternalAccessible := 'False'; ExternalVisible := 'False'; ExternalWritable := 'False'} : UInt;
      弹窗Temp : Array[1..10] of Int;
      AlarmID : Int;
      TON { S7_SetPoint := 'True'} : Array[0..10] of TON_TIME;
      TOF { S7_SetPoint := 'True'} : Array[0..10] of TOF_TIME;
      sUP { S7_SetPoint := 'True'} : Array[0..10] of Bool;
      更新RFID完成 : Bool;
   END_VAR
   VAR_TEMP
      Tempresult : USInt;
      本站站号乘10 : UInt;
   END_VAR
   // // TON[0] : 托盘流入1托盘到位传感器 / iA-Rotating product Check
   // // TON[1] : 托盘流入1托盘到位传感器
   // // TON[2] : 托盘流入1产品有无传感器
   // // TON[3] : 托盘流入1产品有无传感器
   // // TON[4] : 托盘流入1姿态检测光电2
   // // TON[5] : 托盘流入1姿态检测光电3
   // // TON[0].Q : 托盘流入1托盘到位 / iA-Rotating product Check
   // // TON[1].Q : 托盘流入1托盘无
   // // TON[2].Q : 托盘流入1有产品
   // // TON[3].Q : 托盘流入1无产品
   // // TON[4].Q : 托盘流入1姿态检测光电2
   // // TON[5].Q : 托盘流入1姿态检测光电3
   // // TOF[1] : iA-Rotating product Check
BEGIN
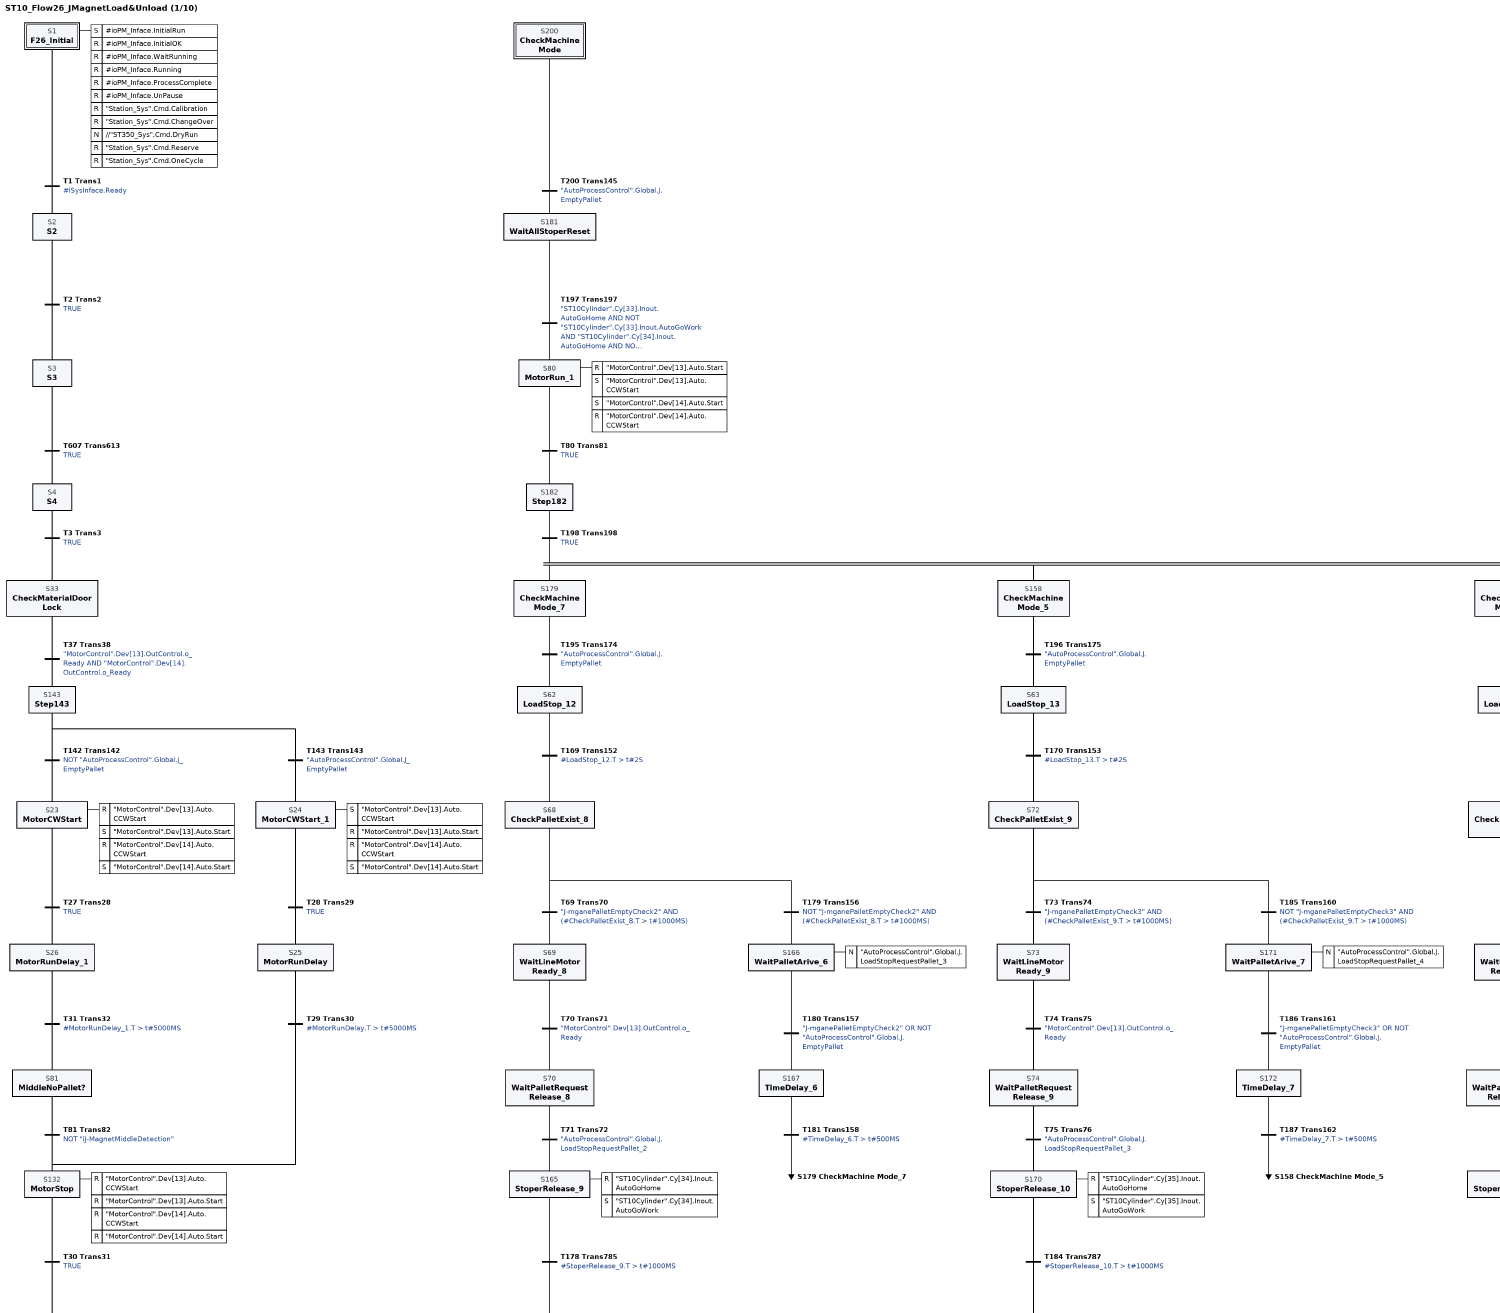
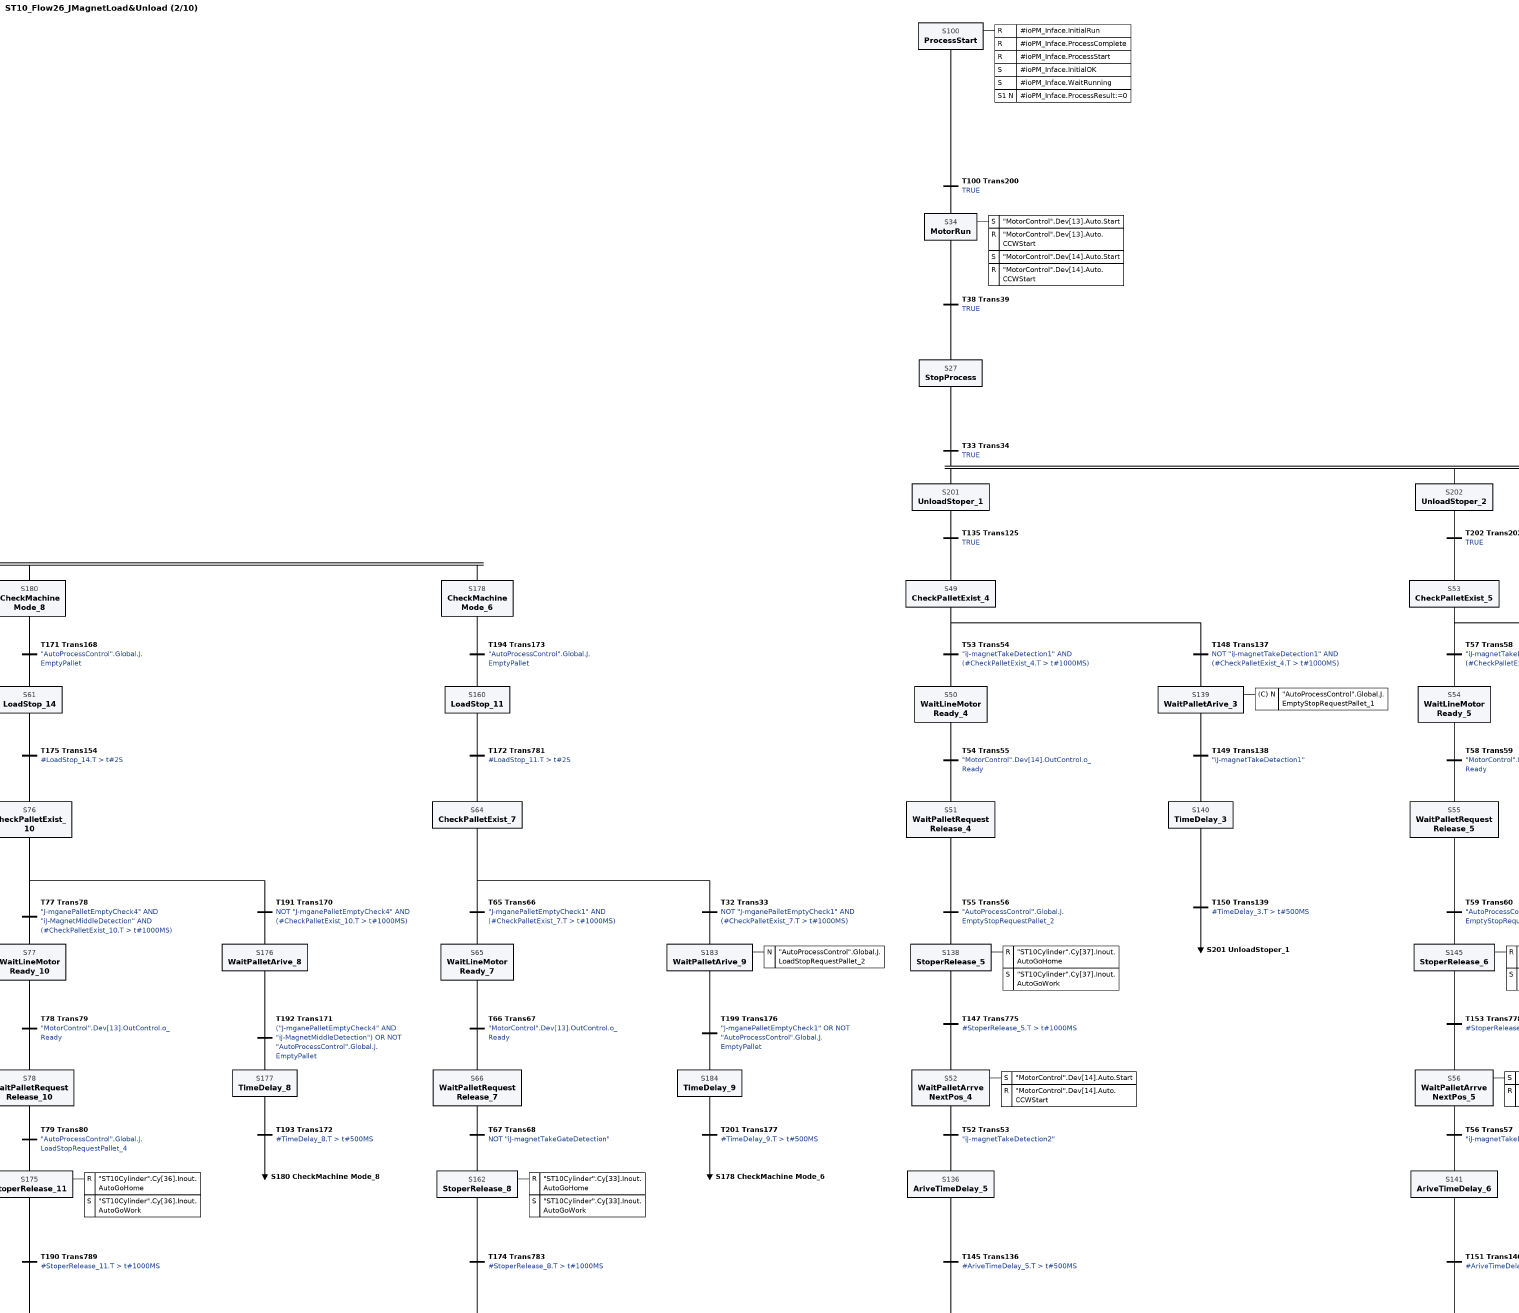
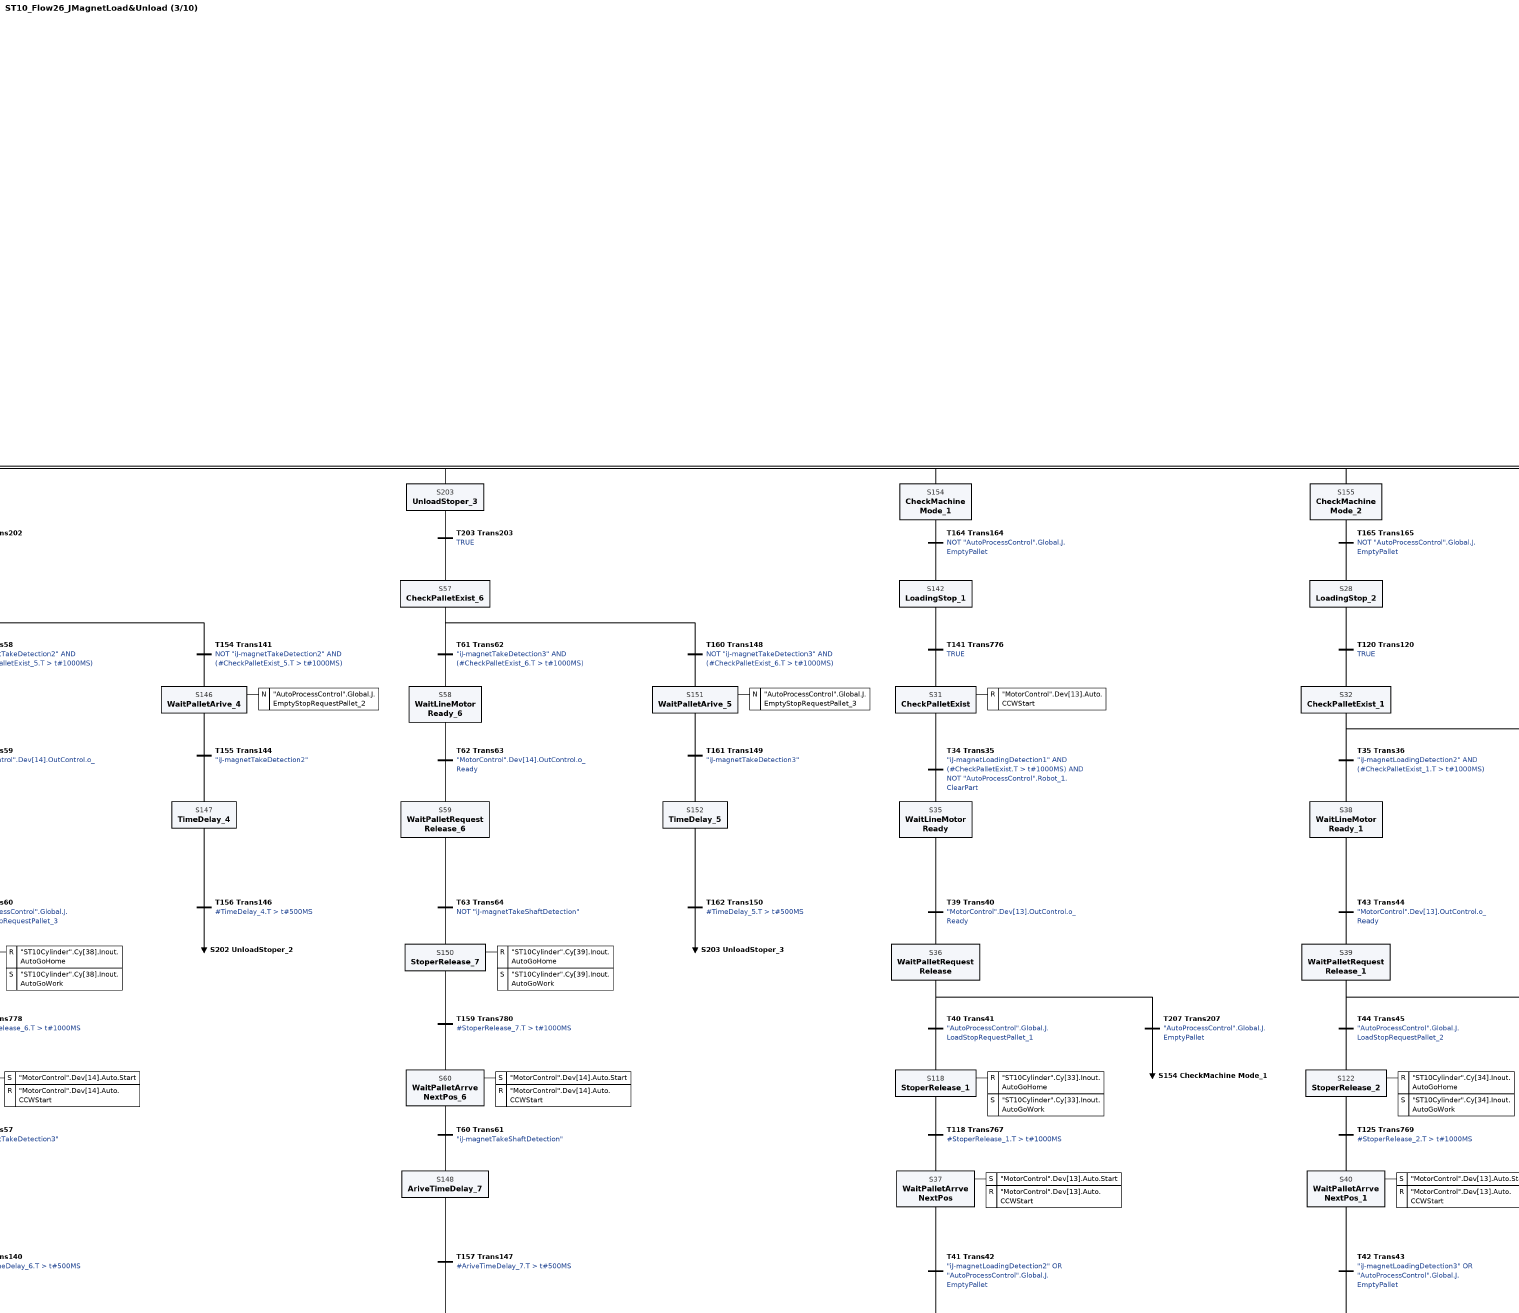
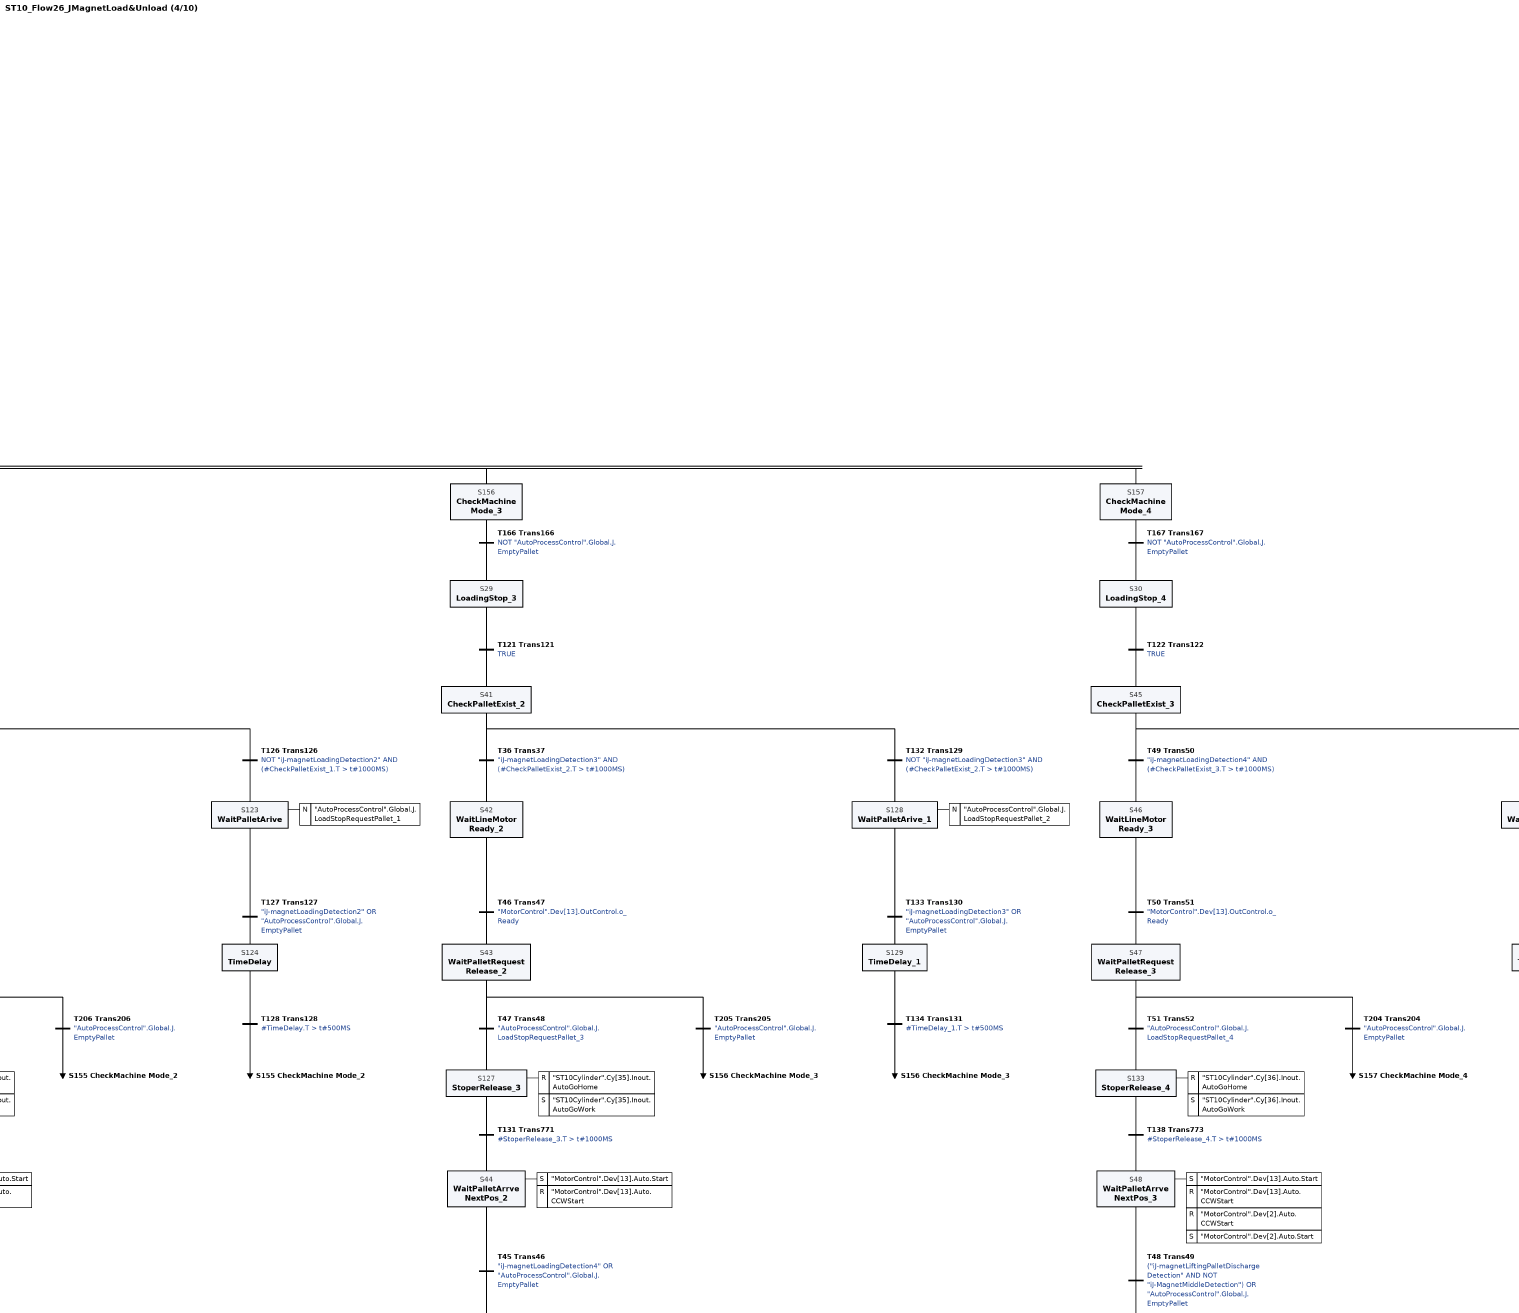
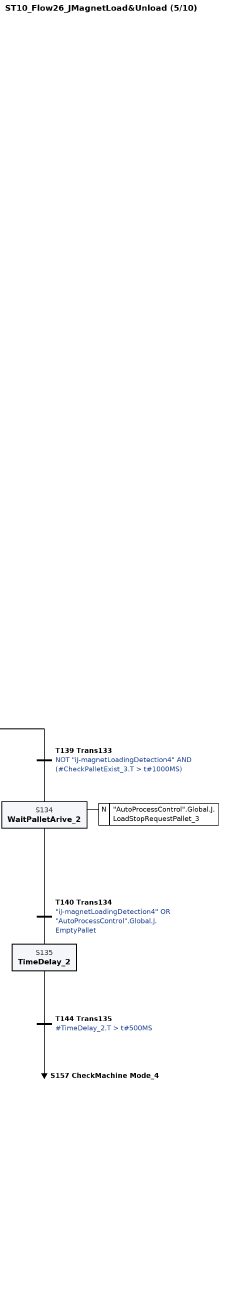
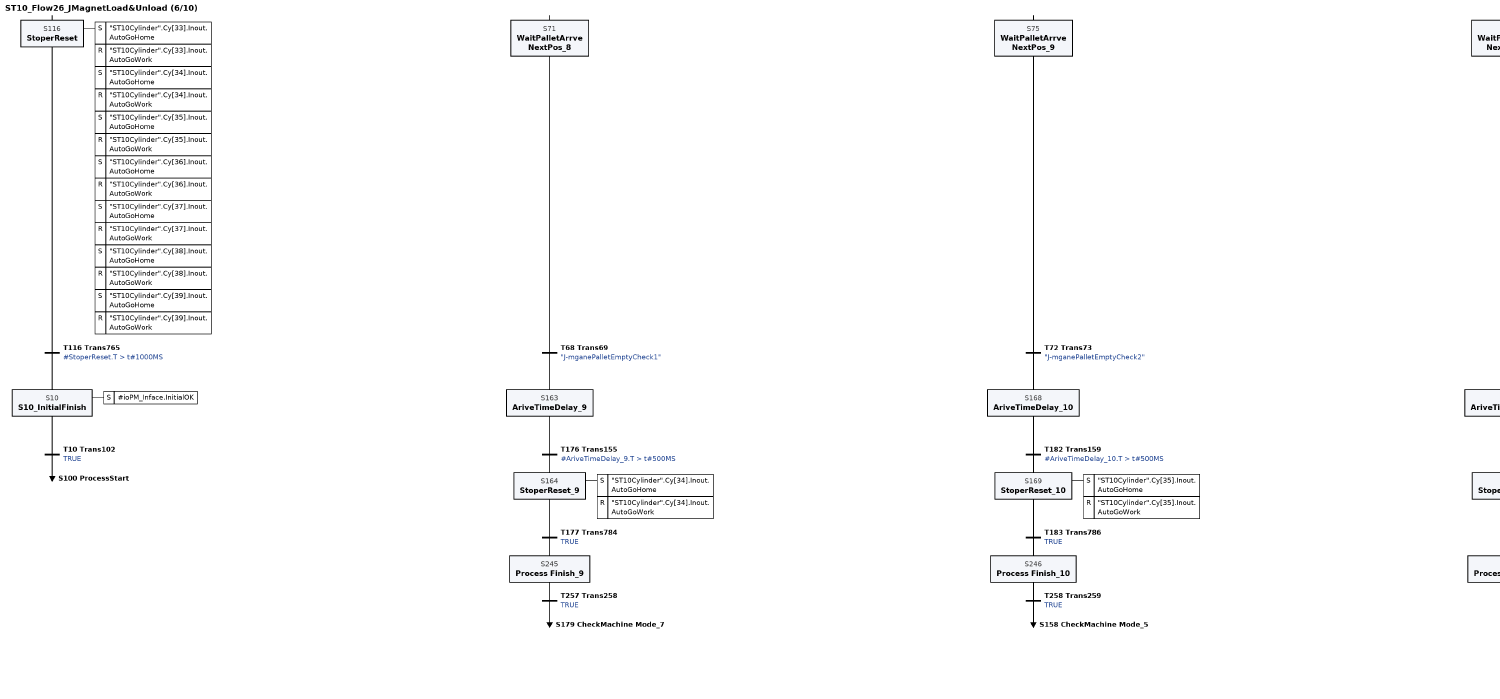
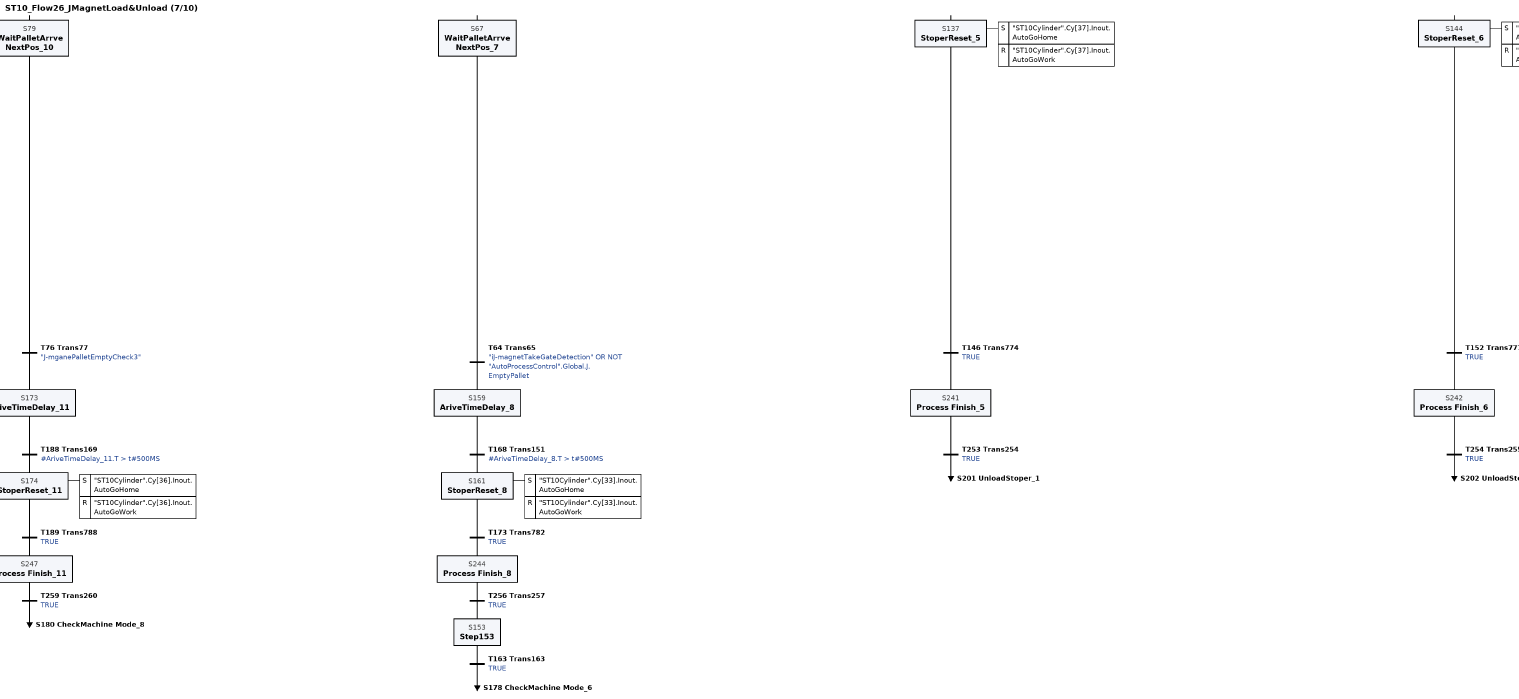
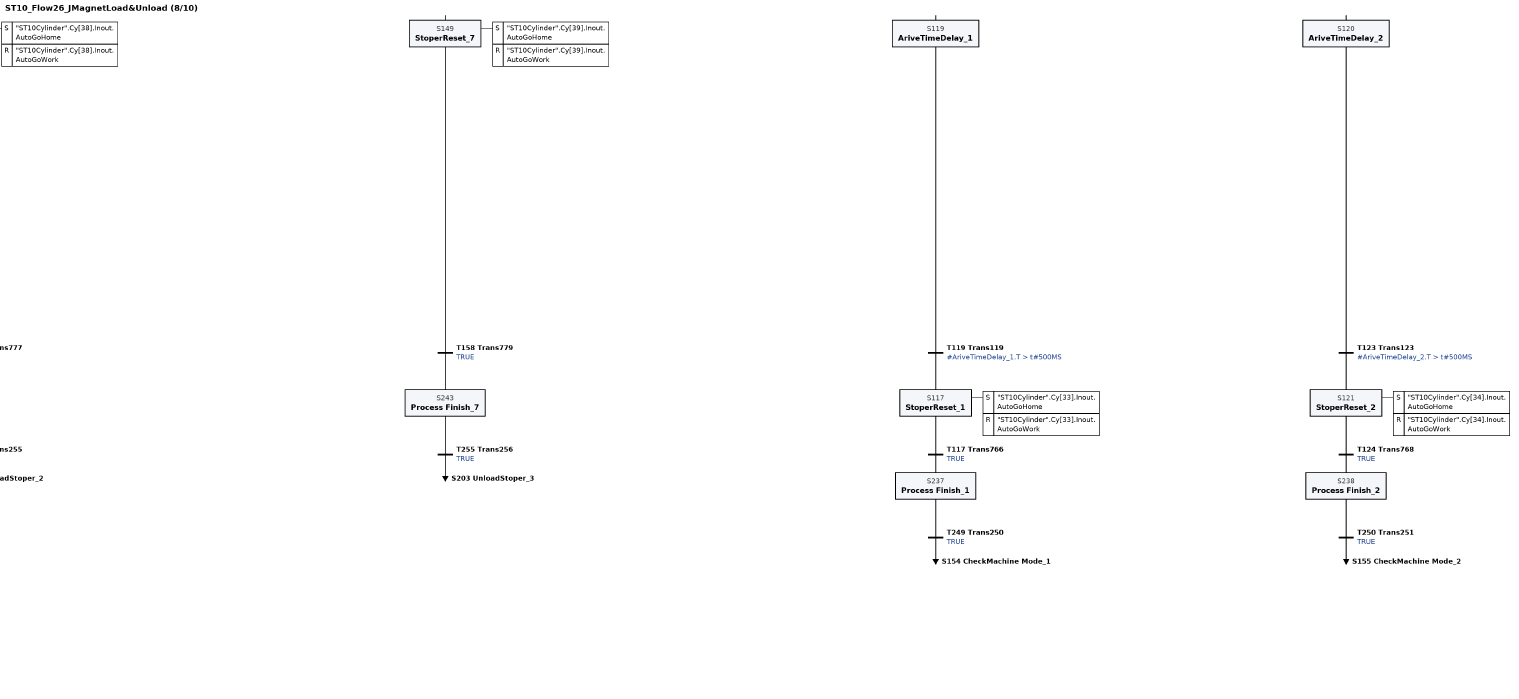
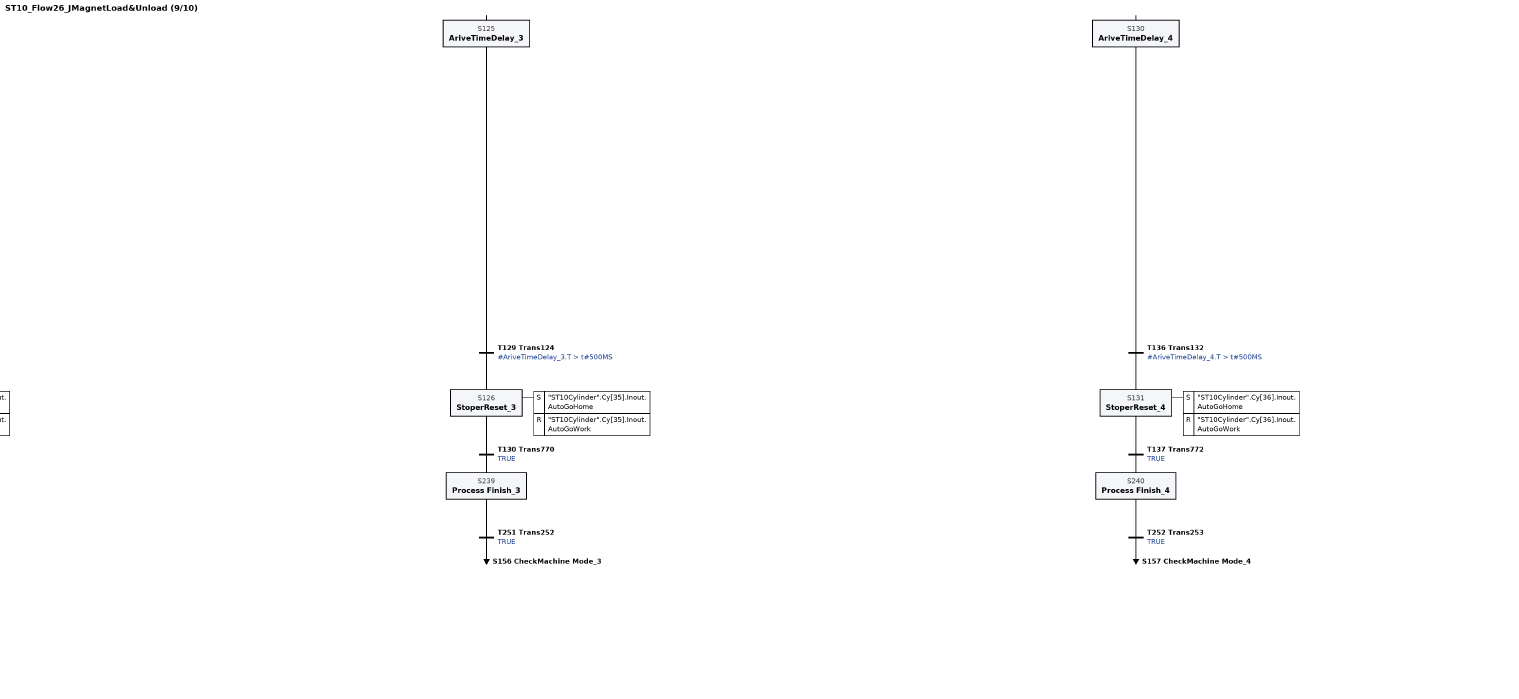
   // permanent pre-instructions
   NETWORK 1
      #TON[10].TON(IN := "AlwaysTRUE" AND "Station_Sys".Alarm.ImmediatelyStop, PT := T#300ms);
      #ioPM_Inface.AlarmImdilyStop := #TON[10].Q;
      #ioPM_Inface.AlarmCycleStop := "AlwaysTRUE" AND "Station_Sys".Alarm.CycleStop;
   NETWORK 2
      IF NOT False THEN
          #sCtrlMode(iSysInface := #iSysInface, ioPM_Inface := #ioPM_Inface, ioGraphCtrl := #RT_DATA.MOP);   // "SysFlowCtrlGraph"
      END_IF;
   NETWORK 3
      #TON[0].TON(IN := "AlwaysTRUE" AND "iJ-magnetLiftingPalletDischargeDetection", PT := t#2000ms);   // 工位11有托盘
      #TOF[1].TOF(IN := "AlwaysTRUE" AND NOT "iJ-magnetLiftingPalletDischargeDetection", PT := T#300ms);   // 工位无托盘
      #TON[2].TON(IN := "AlwaysTRUE", PT := T#300ms);
      #TOF[3].TOF(IN := "AlwaysTRUE", PT := T#300ms);
      #TON[4].TON(IN := "AlwaysTRUE", PT := T#300ms);
      #TOF[5].TOF(IN := "AlwaysTRUE", PT := T#300ms);
   NETWORK 4
      #前站站号 := 345;
      #本站站号 := 350;

   // sequencer 1: S01-S99 初始化 / S01-S99 Initial
   INITIAL_STEP F26_Initial:   // S1, max time T#10S, warning time T#7S
              S    #ioPM_Inface.InitialRun
              R    #ioPM_Inface.InitialOK
              R    #ioPM_Inface.WaitRunning
              R    #ioPM_Inface.Running
              R    #ioPM_Inface.ProcessComplete
              R    #ioPM_Inface.UnPause
              R    "Station_Sys".Cmd.Calibration
              R    "Station_Sys".Cmd.ChangeOver
                   //"ST350_Sys".Cmd.DryRun
              R    "Station_Sys".Cmd.Reserve
              R    "Station_Sys".Cmd.OneCycle
   END_STEP
   TRANSITION Trans1 FROM F26_Initial TO S2   // T1
      := #iSysInface.Ready;
   END_TRANSITION
   STEP S2:   // S2, max time T#10S, warning time T#7S
   END_STEP
   TRANSITION Trans2 FROM S2 TO S3   // T2
      := TRUE;
   END_TRANSITION
   STEP S4:   // S4, max time T#10S, warning time T#7S
   END_STEP
   TRANSITION Trans3 FROM S4 TO CheckMaterialDoorLock   // T3
      := TRUE;
   END_TRANSITION
   STEP MotorRunDelay_1:   // S26, max time T#10S, warning time T#7S
   END_STEP
   TRANSITION Trans32 FROM MotorRunDelay_1 TO "MiddleNoPallet?"   // T31
      := #MotorRunDelay_1.T > t#5000MS;
   END_TRANSITION
   STEP S10_InitialFinish:   // S10, max time T#10S, warning time T#7S
              S    #ioPM_Inface.InitialOK
   END_STEP
   TRANSITION Trans102 FROM S10_InitialFinish TO ProcessStart   // T10, jump
      := TRUE;
   END_TRANSITION
   STEP S3:   // S3, max time T#10S, warning time T#7S
   END_STEP
   TRANSITION Trans613 FROM S3 TO S4   // T607
      := TRUE;
   END_TRANSITION
   STEP CheckMaterialDoorLock:   // S33, max time T#10S, warning time T#7S
   END_STEP
   TRANSITION Trans38 FROM CheckMaterialDoorLock TO Step143   // T37
      := "MotorControl".Dev[13].OutControl.o_Ready AND "MotorControl".Dev[14].OutControl.o_Ready;
   END_TRANSITION
   STEP "MiddleNoPallet?":   // S81, max time T#10S, warning time T#7S
   END_STEP
   TRANSITION Trans82 FROM "MiddleNoPallet?" TO MotorStop   // T81
      := NOT "iJ-MagnetMiddleDetection";
   END_TRANSITION
   STEP StoperReset:   // S116, max time T#10S, warning time T#7S
              S    "ST10Cylinder".Cy[33].Inout.AutoGoHome
              R    "ST10Cylinder".Cy[33].Inout.AutoGoWork
              S    "ST10Cylinder".Cy[34].Inout.AutoGoHome
              R    "ST10Cylinder".Cy[34].Inout.AutoGoWork
              S    "ST10Cylinder".Cy[35].Inout.AutoGoHome
              R    "ST10Cylinder".Cy[35].Inout.AutoGoWork
              S    "ST10Cylinder".Cy[36].Inout.AutoGoHome
              R    "ST10Cylinder".Cy[36].Inout.AutoGoWork
              S    "ST10Cylinder".Cy[37].Inout.AutoGoHome
              R    "ST10Cylinder".Cy[37].Inout.AutoGoWork
              S    "ST10Cylinder".Cy[38].Inout.AutoGoHome
              R    "ST10Cylinder".Cy[38].Inout.AutoGoWork
              S    "ST10Cylinder".Cy[39].Inout.AutoGoHome
              R    "ST10Cylinder".Cy[39].Inout.AutoGoWork
   END_STEP
   TRANSITION Trans765 FROM StoperReset TO S10_InitialFinish   // T116
      := #StoperReset.T > t#1000MS;
   END_TRANSITION
   STEP MotorCWStart_1:   // S24, max time T#10S, warning time T#7S
              S    "MotorControl".Dev[13].Auto.CCWStart
              R    "MotorControl".Dev[13].Auto.Start
              R    "MotorControl".Dev[14].Auto.CCWStart
              S    "MotorControl".Dev[14].Auto.Start
   END_STEP
   TRANSITION Trans29 FROM MotorCWStart_1 TO MotorRunDelay   // T28
      := TRUE;
   END_TRANSITION
   STEP Step143:   // S143, max time T#10S, warning time T#7S
   END_STEP
   TRANSITION Trans142 FROM Step143 TO MotorCWStart   // T142
      := NOT "AutoProcessControl".Global.J_EmptyPallet;
   END_TRANSITION
   TRANSITION Trans143 FROM Step143 TO MotorCWStart_1   // T143
      := "AutoProcessControl".Global.J_EmptyPallet;
   END_TRANSITION
   STEP MotorCWStart:   // S23, max time T#10S, warning time T#7S
              R    "MotorControl".Dev[13].Auto.CCWStart
              S    "MotorControl".Dev[13].Auto.Start
              R    "MotorControl".Dev[14].Auto.CCWStart
              S    "MotorControl".Dev[14].Auto.Start
   END_STEP
   TRANSITION Trans28 FROM MotorCWStart TO MotorRunDelay_1   // T27
      := TRUE;
   END_TRANSITION
   STEP MotorStop:   // S132, max time T#10S, warning time T#7S
              R    "MotorControl".Dev[13].Auto.CCWStart
              R    "MotorControl".Dev[13].Auto.Start
              R    "MotorControl".Dev[14].Auto.CCWStart
              R    "MotorControl".Dev[14].Auto.Start
   END_STEP
   TRANSITION Trans31 FROM MotorStop TO StoperReset   // T30
      := TRUE;
   END_TRANSITION
   STEP MotorRunDelay:   // S25, max time T#10S, warning time T#7S
   END_STEP
   TRANSITION Trans30 FROM MotorRunDelay TO MotorStop   // T29
      := #MotorRunDelay.T > t#5000MS;
   END_TRANSITION

   // sequencer 2: S100-S199 等待到位 / S100-S199 CheckLineMode
   STEP ProcessStart:   // S100, max time T#10S, warning time T#7S
      // 自动等待开始运行
              R    #ioPM_Inface.InitialRun
              R    #ioPM_Inface.ProcessComplete
              R    #ioPM_Inface.ProcessStart
              S    #ioPM_Inface.InitialOK
              S    #ioPM_Inface.WaitRunning
          S1  N    #ioPM_Inface.ProcessResult:=0
   END_STEP
   TRANSITION Trans200 FROM ProcessStart TO MotorRun   // T100
      := TRUE;
   END_TRANSITION
   STEP "Process Finish_1":   // S237, max time T#10S, warning time T#7S
   END_STEP
   TRANSITION Trans250 FROM "Process Finish_1" TO "CheckMachine Mode_1"   // T249, jump
      := TRUE;
   END_TRANSITION
   STEP StopProcess:   // S27, max time T#10S, warning time T#7S
   END_STEP
   TRANSITION Trans34 FROM StopProcess TO (UnloadStoper_1, UnloadStoper_2, UnloadStoper_3, "CheckMachine Mode_1", "CheckMachine Mode_2", "CheckMachine Mode_3", "CheckMachine Mode_4")   // T33
      := TRUE;
   END_TRANSITION
   STEP MotorRun:   // S34, max time T#10S, warning time T#7S
              S    "MotorControl".Dev[13].Auto.Start
              R    "MotorControl".Dev[13].Auto.CCWStart
              S    "MotorControl".Dev[14].Auto.Start
              R    "MotorControl".Dev[14].Auto.CCWStart
   END_STEP
   TRANSITION Trans39 FROM MotorRun TO StopProcess   // T38
      := TRUE;
   END_TRANSITION
   STEP LoadingStop_4:   // S30, max time T#10S, warning time T#7S
   END_STEP
   TRANSITION Trans122 FROM LoadingStop_4 TO CheckPalletExist_3   // T122
      := TRUE;
   END_TRANSITION
   STEP LoadingStop_2:   // S28, max time T#10S, warning time T#7S
   END_STEP
   TRANSITION Trans120 FROM LoadingStop_2 TO CheckPalletExist_1   // T120
      := TRUE;
   END_TRANSITION
   STEP "CheckMachine Mode_3":   // S156, max time T#10S, warning time T#7S
   END_STEP
   TRANSITION Trans166 FROM "CheckMachine Mode_3" TO LoadingStop_3   // T166
      := NOT "AutoProcessControl".Global.J.EmptyPallet;
   END_TRANSITION
   STEP LoadingStop_3:   // S29, max time T#10S, warning time T#7S
   END_STEP
   TRANSITION Trans121 FROM LoadingStop_3 TO CheckPalletExist_2   // T121
      := TRUE;
   END_TRANSITION
   STEP CheckPalletExist:   // S31, max time T#10S, warning time T#7S
              R    "MotorControl".Dev[13].Auto.CCWStart
   END_STEP
   TRANSITION Trans35 FROM CheckPalletExist TO WaitLineMotorReady   // T34
      := "iJ-magnetLoadingDetection1" AND (#CheckPalletExist.T > t#1000MS) AND NOT "AutoProcessControl".Robot_1.ClearPart;
   END_TRANSITION
   STEP AriveTimeDelay_1:   // S119, max time T#10S, warning time T#7S
   END_STEP
   TRANSITION Trans119 FROM AriveTimeDelay_1 TO StoperReset_1   // T119
      := #AriveTimeDelay_1.T > t#500MS;
   END_TRANSITION
   STEP WaitLineMotorReady:   // S35, max time T#10S, warning time T#7S
   END_STEP
   TRANSITION Trans40 FROM WaitLineMotorReady TO WaitPalletRequestRelease   // T39
      := "MotorControl".Dev[13].OutControl.o_Ready;
   END_TRANSITION
   STEP WaitPalletRequestRelease:   // S36, max time T#10S, warning time T#7S
   END_STEP
   TRANSITION Trans41 FROM WaitPalletRequestRelease TO StoperRelease_1   // T40
      := "AutoProcessControl".Global.J.LoadStopRequestPallet_1;
   END_TRANSITION
   TRANSITION Trans207 FROM WaitPalletRequestRelease TO "CheckMachine Mode_1"   // T207, jump
      := "AutoProcessControl".Global.J.EmptyPallet;
   END_TRANSITION
   STEP LoadingStop_1:   // S142, max time T#10S, warning time T#7S
   END_STEP
   TRANSITION Trans776 FROM LoadingStop_1 TO CheckPalletExist   // T141
      := TRUE;
   END_TRANSITION
   STEP WaitPalletArrveNextPos:   // S37, max time T#10S, warning time T#7S
              S    "MotorControl".Dev[13].Auto.Start
              R    "MotorControl".Dev[13].Auto.CCWStart
   END_STEP
   TRANSITION Trans42 FROM WaitPalletArrveNextPos TO AriveTimeDelay_1   // T41
      := "iJ-magnetLoadingDetection2" OR "AutoProcessControl".Global.J.EmptyPallet;
   END_TRANSITION
   STEP "Process Finish_2":   // S238, max time T#10S, warning time T#7S
   END_STEP
   TRANSITION Trans251 FROM "Process Finish_2" TO "CheckMachine Mode_2"   // T250, jump
      := TRUE;
   END_TRANSITION
   STEP StoperReset_1:   // S117, max time T#10S, warning time T#7S
              S    "ST10Cylinder".Cy[33].Inout.AutoGoHome
              R    "ST10Cylinder".Cy[33].Inout.AutoGoWork
   END_STEP
   TRANSITION Trans766 FROM StoperReset_1 TO "Process Finish_1"   // T117
      := TRUE;
   END_TRANSITION
   STEP StoperRelease_1:   // S118, max time T#10S, warning time T#7S
              R    "ST10Cylinder".Cy[33].Inout.AutoGoHome
              S    "ST10Cylinder".Cy[33].Inout.AutoGoWork
   END_STEP
   TRANSITION Trans767 FROM StoperRelease_1 TO WaitPalletArrveNextPos   // T118
      := #StoperRelease_1.T > t#1000MS;
   END_TRANSITION
   STEP CheckPalletExist_1:   // S32, max time T#10S, warning time T#7S
   END_STEP
   TRANSITION Trans36 FROM CheckPalletExist_1 TO WaitLineMotorReady_1   // T35
      := "iJ-magnetLoadingDetection2" AND (#CheckPalletExist_1.T > t#1000MS);
   END_TRANSITION
   TRANSITION Trans126 FROM CheckPalletExist_1 TO WaitPalletArive   // T126
      := NOT "iJ-magnetLoadingDetection2" AND (#CheckPalletExist_1.T > t#1000MS);
   END_TRANSITION
   STEP AriveTimeDelay_2:   // S120, max time T#10S, warning time T#7S
   END_STEP
   TRANSITION Trans123 FROM AriveTimeDelay_2 TO StoperReset_2   // T123
      := #AriveTimeDelay_2.T > t#500MS;
   END_TRANSITION
   STEP WaitLineMotorReady_1:   // S38, max time T#10S, warning time T#7S
   END_STEP
   TRANSITION Trans44 FROM WaitLineMotorReady_1 TO WaitPalletRequestRelease_1   // T43
      := "MotorControl".Dev[13].OutControl.o_Ready;
   END_TRANSITION
   STEP WaitPalletRequestRelease_1:   // S39, max time T#10S, warning time T#7S
   END_STEP
   TRANSITION Trans45 FROM WaitPalletRequestRelease_1 TO StoperRelease_2   // T44
      := "AutoProcessControl".Global.J.LoadStopRequestPallet_2;
   END_TRANSITION
   TRANSITION Trans206 FROM WaitPalletRequestRelease_1 TO "CheckMachine Mode_2"   // T206, jump
      := "AutoProcessControl".Global.J.EmptyPallet;
   END_TRANSITION
   STEP WaitPalletArrveNextPos_1:   // S40, max time T#10S, warning time T#7S
              S    "MotorControl".Dev[13].Auto.Start
              R    "MotorControl".Dev[13].Auto.CCWStart
   END_STEP
   TRANSITION Trans43 FROM WaitPalletArrveNextPos_1 TO AriveTimeDelay_2   // T42
      := "iJ-magnetLoadingDetection3" OR "AutoProcessControl".Global.J.EmptyPallet;
   END_TRANSITION
   STEP StoperReset_2:   // S121, max time T#10S, warning time T#7S
              S    "ST10Cylinder".Cy[34].Inout.AutoGoHome
              R    "ST10Cylinder".Cy[34].Inout.AutoGoWork
   END_STEP
   TRANSITION Trans768 FROM StoperReset_2 TO "Process Finish_2"   // T124
      := TRUE;
   END_TRANSITION
   STEP StoperRelease_2:   // S122, max time T#10S, warning time T#7S
              R    "ST10Cylinder".Cy[34].Inout.AutoGoHome
              S    "ST10Cylinder".Cy[34].Inout.AutoGoWork
   END_STEP
   TRANSITION Trans769 FROM StoperRelease_2 TO WaitPalletArrveNextPos_1   // T125
      := #StoperRelease_2.T > t#1000MS;
   END_TRANSITION
   STEP WaitPalletArive:   // S123, max time T#10S, warning time T#7S
              N    "AutoProcessControl".Global.J.LoadStopRequestPallet_1
   END_STEP
   TRANSITION Trans127 FROM WaitPalletArive TO TimeDelay   // T127
      := "iJ-magnetLoadingDetection2" OR "AutoProcessControl".Global.J.EmptyPallet;
   END_TRANSITION
   STEP TimeDelay:   // S124, max time T#10S, warning time T#7S
   END_STEP
   TRANSITION Trans128 FROM TimeDelay TO "CheckMachine Mode_2"   // T128, jump
      := #TimeDelay.T > t#500MS;
   END_TRANSITION
   STEP "Process Finish_3":   // S239, max time T#10S, warning time T#7S
   END_STEP
   TRANSITION Trans252 FROM "Process Finish_3" TO "CheckMachine Mode_3"   // T251, jump
      := TRUE;
   END_TRANSITION
   STEP CheckPalletExist_2:   // S41, max time T#10S, warning time T#7S
   END_STEP
   TRANSITION Trans37 FROM CheckPalletExist_2 TO WaitLineMotorReady_2   // T36
      := "iJ-magnetLoadingDetection3" AND (#CheckPalletExist_2.T > t#1000MS);
   END_TRANSITION
   TRANSITION Trans129 FROM CheckPalletExist_2 TO WaitPalletArive_1   // T132
      := NOT "iJ-magnetLoadingDetection3" AND (#CheckPalletExist_2.T > t#1000MS);
   END_TRANSITION
   STEP AriveTimeDelay_3:   // S125, max time T#10S, warning time T#7S
   END_STEP
   TRANSITION Trans124 FROM AriveTimeDelay_3 TO StoperReset_3   // T129
      := #AriveTimeDelay_3.T > t#500MS;
   END_TRANSITION
   STEP WaitLineMotorReady_2:   // S42, max time T#10S, warning time T#7S
   END_STEP
   TRANSITION Trans47 FROM WaitLineMotorReady_2 TO WaitPalletRequestRelease_2   // T46
      := "MotorControl".Dev[13].OutControl.o_Ready;
   END_TRANSITION
   STEP WaitPalletRequestRelease_2:   // S43, max time T#10S, warning time T#7S
   END_STEP
   TRANSITION Trans48 FROM WaitPalletRequestRelease_2 TO StoperRelease_3   // T47
      := "AutoProcessControl".Global.J.LoadStopRequestPallet_3;
   END_TRANSITION
   TRANSITION Trans205 FROM WaitPalletRequestRelease_2 TO "CheckMachine Mode_3"   // T205, jump
      := "AutoProcessControl".Global.J.EmptyPallet;
   END_TRANSITION
   STEP WaitPalletArrveNextPos_2:   // S44, max time T#10S, warning time T#7S
              S    "MotorControl".Dev[13].Auto.Start
              R    "MotorControl".Dev[13].Auto.CCWStart
   END_STEP
   TRANSITION Trans46 FROM WaitPalletArrveNextPos_2 TO AriveTimeDelay_3   // T45
      := "iJ-magnetLoadingDetection4" OR "AutoProcessControl".Global.J.EmptyPallet;
   END_TRANSITION
   STEP StoperReset_3:   // S126, max time T#10S, warning time T#7S
              S    "ST10Cylinder".Cy[35].Inout.AutoGoHome
              R    "ST10Cylinder".Cy[35].Inout.AutoGoWork
   END_STEP
   TRANSITION Trans770 FROM StoperReset_3 TO "Process Finish_3"   // T130
      := TRUE;
   END_TRANSITION
   STEP StoperRelease_3:   // S127, max time T#10S, warning time T#7S
              R    "ST10Cylinder".Cy[35].Inout.AutoGoHome
              S    "ST10Cylinder".Cy[35].Inout.AutoGoWork
   END_STEP
   TRANSITION Trans771 FROM StoperRelease_3 TO WaitPalletArrveNextPos_2   // T131
      := #StoperRelease_3.T > t#1000MS;
   END_TRANSITION
   STEP WaitPalletArive_1:   // S128, max time T#10S, warning time T#7S
              N    "AutoProcessControl".Global.J.LoadStopRequestPallet_2
   END_STEP
   TRANSITION Trans130 FROM WaitPalletArive_1 TO TimeDelay_1   // T133
      := "iJ-magnetLoadingDetection3" OR "AutoProcessControl".Global.J.EmptyPallet;
   END_TRANSITION
   STEP TimeDelay_1:   // S129, max time T#10S, warning time T#7S
   END_STEP
   TRANSITION Trans131 FROM TimeDelay_1 TO "CheckMachine Mode_3"   // T134, jump
      := #TimeDelay_1.T > t#500MS;
   END_TRANSITION
   STEP UnloadStoper_1:   // S201, max time T#10S, warning time T#7S
   END_STEP
   TRANSITION Trans125 FROM UnloadStoper_1 TO CheckPalletExist_4   // T135
      := TRUE;
   END_TRANSITION
   STEP "Process Finish_4":   // S240, max time T#10S, warning time T#7S
   END_STEP
   TRANSITION Trans253 FROM "Process Finish_4" TO "CheckMachine Mode_4"   // T252, jump
      := TRUE;
   END_TRANSITION
   STEP CheckPalletExist_3:   // S45, max time T#10S, warning time T#7S
   END_STEP
   TRANSITION Trans50 FROM CheckPalletExist_3 TO WaitLineMotorReady_3   // T49
      := "iJ-magnetLoadingDetection4" AND (#CheckPalletExist_3.T > t#1000MS);
   END_TRANSITION
   TRANSITION Trans133 FROM CheckPalletExist_3 TO WaitPalletArive_2   // T139
      := NOT "iJ-magnetLoadingDetection4" AND (#CheckPalletExist_3.T > t#1000MS);
   END_TRANSITION
   STEP AriveTimeDelay_4:   // S130, max time T#10S, warning time T#7S
   END_STEP
   TRANSITION Trans132 FROM AriveTimeDelay_4 TO StoperReset_4   // T136
      := #AriveTimeDelay_4.T > t#500MS;
   END_TRANSITION
   STEP WaitLineMotorReady_3:   // S46, max time T#10S, warning time T#7S
   END_STEP
   TRANSITION Trans51 FROM WaitLineMotorReady_3 TO WaitPalletRequestRelease_3   // T50
      := "MotorControl".Dev[13].OutControl.o_Ready;
   END_TRANSITION
   STEP WaitPalletRequestRelease_3:   // S47, max time T#10S, warning time T#7S
   END_STEP
   TRANSITION Trans52 FROM WaitPalletRequestRelease_3 TO StoperRelease_4   // T51
      := "AutoProcessControl".Global.J.LoadStopRequestPallet_4;
   END_TRANSITION
   TRANSITION Trans204 FROM WaitPalletRequestRelease_3 TO "CheckMachine Mode_4"   // T204, jump
      := "AutoProcessControl".Global.J.EmptyPallet;
   END_TRANSITION
   STEP WaitPalletArrveNextPos_3:   // S48, max time T#10S, warning time T#7S
              S    "MotorControl".Dev[13].Auto.Start
              R    "MotorControl".Dev[13].Auto.CCWStart
              R    "MotorControl".Dev[2].Auto.CCWStart
              S    "MotorControl".Dev[2].Auto.Start
   END_STEP
   TRANSITION Trans49 FROM WaitPalletArrveNextPos_3 TO AriveTimeDelay_4   // T48
      := ("iJ-magnetLiftingPalletDischargeDetection" AND NOT "iJ-MagnetMiddleDetection") OR "AutoProcessControl".Global.J.EmptyPallet;
   END_TRANSITION
   STEP StoperReset_4:   // S131, max time T#10S, warning time T#7S
              S    "ST10Cylinder".Cy[36].Inout.AutoGoHome
              R    "ST10Cylinder".Cy[36].Inout.AutoGoWork
   END_STEP
   TRANSITION Trans772 FROM StoperReset_4 TO "Process Finish_4"   // T137
      := TRUE;
   END_TRANSITION
   STEP StoperRelease_4:   // S133, max time T#10S, warning time T#7S
              R    "ST10Cylinder".Cy[36].Inout.AutoGoHome
              S    "ST10Cylinder".Cy[36].Inout.AutoGoWork
   END_STEP
   TRANSITION Trans773 FROM StoperRelease_4 TO WaitPalletArrveNextPos_3   // T138
      := #StoperRelease_4.T > t#1000MS;
   END_TRANSITION
   STEP WaitPalletArive_2:   // S134, max time T#10S, warning time T#7S
              N    "AutoProcessControl".Global.J.LoadStopRequestPallet_3
   END_STEP
   TRANSITION Trans134 FROM WaitPalletArive_2 TO TimeDelay_2   // T140
      := "iJ-magnetLoadingDetection4" OR "AutoProcessControl".Global.J.EmptyPallet;
   END_TRANSITION
   STEP TimeDelay_2:   // S135, max time T#10S, warning time T#7S
   END_STEP
   TRANSITION Trans135 FROM TimeDelay_2 TO "CheckMachine Mode_4"   // T144, jump
      := #TimeDelay_2.T > t#500MS;
   END_TRANSITION
   STEP UnloadStoper_2:   // S202, max time T#10S, warning time T#7S
   END_STEP
   TRANSITION Trans202 FROM UnloadStoper_2 TO CheckPalletExist_5   // T202
      := TRUE;
   END_TRANSITION
   STEP UnloadStoper_3:   // S203, max time T#10S, warning time T#7S
   END_STEP
   TRANSITION Trans203 FROM UnloadStoper_3 TO CheckPalletExist_6   // T203
      := TRUE;
   END_TRANSITION
   STEP "Process Finish_6":   // S242, max time T#10S, warning time T#7S
   END_STEP
   TRANSITION Trans255 FROM "Process Finish_6" TO UnloadStoper_2   // T254, jump
      := TRUE;
   END_TRANSITION
   STEP "Process Finish_5":   // S241, max time T#10S, warning time T#7S
   END_STEP
   TRANSITION Trans254 FROM "Process Finish_5" TO UnloadStoper_1   // T253, jump
      := TRUE;
   END_TRANSITION
   STEP CheckPalletExist_4:   // S49, max time T#10S, warning time T#7S
   END_STEP
   TRANSITION Trans54 FROM CheckPalletExist_4 TO WaitLineMotorReady_4   // T53
      := "iJ-magnetTakeDetection1" AND (#CheckPalletExist_4.T > t#1000MS);
   END_TRANSITION
   TRANSITION Trans137 FROM CheckPalletExist_4 TO WaitPalletArive_3   // T148
      := NOT "iJ-magnetTakeDetection1" AND (#CheckPalletExist_4.T > t#1000MS);
   END_TRANSITION
   STEP AriveTimeDelay_5:   // S136, max time T#10S, warning time T#7S
   END_STEP
   TRANSITION Trans136 FROM AriveTimeDelay_5 TO StoperReset_5   // T145
      := #AriveTimeDelay_5.T > t#500MS;
   END_TRANSITION
   STEP WaitLineMotorReady_4:   // S50, max time T#10S, warning time T#7S
   END_STEP
   TRANSITION Trans55 FROM WaitLineMotorReady_4 TO WaitPalletRequestRelease_4   // T54
      := "MotorControl".Dev[14].OutControl.o_Ready;
   END_TRANSITION
   STEP WaitPalletRequestRelease_4:   // S51, max time T#10S, warning time T#7S
   END_STEP
   TRANSITION Trans56 FROM WaitPalletRequestRelease_4 TO StoperRelease_5   // T55
      := "AutoProcessControl".Global.J.EmptyStopRequestPallet_2;
   END_TRANSITION
   STEP WaitPalletArrveNextPos_4:   // S52, max time T#10S, warning time T#7S
              S    "MotorControl".Dev[14].Auto.Start
              R    "MotorControl".Dev[14].Auto.CCWStart
   END_STEP
   TRANSITION Trans53 FROM WaitPalletArrveNextPos_4 TO AriveTimeDelay_5   // T52
      := "iJ-magnetTakeDetection2";
   END_TRANSITION
   STEP StoperReset_5:   // S137, max time T#10S, warning time T#7S
              S    "ST10Cylinder".Cy[37].Inout.AutoGoHome
              R    "ST10Cylinder".Cy[37].Inout.AutoGoWork
   END_STEP
   TRANSITION Trans774 FROM StoperReset_5 TO "Process Finish_5"   // T146
      := TRUE;
   END_TRANSITION
   STEP StoperRelease_5:   // S138, max time T#10S, warning time T#7S
              R    "ST10Cylinder".Cy[37].Inout.AutoGoHome
              S    "ST10Cylinder".Cy[37].Inout.AutoGoWork
   END_STEP
   TRANSITION Trans775 FROM StoperRelease_5 TO WaitPalletArrveNextPos_4   // T147
      := #StoperRelease_5.T > t#1000MS;
   END_TRANSITION
   STEP WaitPalletArive_3:   // S139, max time T#10S, warning time T#7S
      interlock C := "ST10Cylinder".Cy[37].Inout.AutoGoHome AND NOT "ST10Cylinder".Cy[37].Inout.AutoGoWork;
      (C)     N    "AutoProcessControl".Global.J.EmptyStopRequestPallet_1
   END_STEP
   TRANSITION Trans138 FROM WaitPalletArive_3 TO TimeDelay_3   // T149
      := "iJ-magnetTakeDetection1";
   END_TRANSITION
   STEP TimeDelay_3:   // S140, max time T#10S, warning time T#7S
   END_STEP
   TRANSITION Trans139 FROM TimeDelay_3 TO UnloadStoper_1   // T150, jump
      := #TimeDelay_3.T > t#500MS;
   END_TRANSITION
   STEP CheckPalletExist_5:   // S53, max time T#10S, warning time T#7S
   END_STEP
   TRANSITION Trans58 FROM CheckPalletExist_5 TO WaitLineMotorReady_5   // T57
      := "iJ-magnetTakeDetection2" AND (#CheckPalletExist_5.T > t#1000MS);
   END_TRANSITION
   TRANSITION Trans141 FROM CheckPalletExist_5 TO WaitPalletArive_4   // T154
      := NOT "iJ-magnetTakeDetection2" AND (#CheckPalletExist_5.T > t#1000MS);
   END_TRANSITION
   STEP AriveTimeDelay_6:   // S141, max time T#10S, warning time T#7S
   END_STEP
   TRANSITION Trans140 FROM AriveTimeDelay_6 TO StoperReset_6   // T151
      := #AriveTimeDelay_6.T > t#500MS;
   END_TRANSITION
   STEP WaitLineMotorReady_5:   // S54, max time T#10S, warning time T#7S
   END_STEP
   TRANSITION Trans59 FROM WaitLineMotorReady_5 TO WaitPalletRequestRelease_5   // T58
      := "MotorControl".Dev[14].OutControl.o_Ready;
   END_TRANSITION
   STEP WaitPalletRequestRelease_5:   // S55, max time T#10S, warning time T#7S
   END_STEP
   TRANSITION Trans60 FROM WaitPalletRequestRelease_5 TO StoperRelease_6   // T59
      := "AutoProcessControl".Global.J.EmptyStopRequestPallet_3;
   END_TRANSITION
   STEP WaitPalletArrveNextPos_5:   // S56, max time T#10S, warning time T#7S
              S    "MotorControl".Dev[14].Auto.Start
              R    "MotorControl".Dev[14].Auto.CCWStart
   END_STEP
   TRANSITION Trans57 FROM WaitPalletArrveNextPos_5 TO AriveTimeDelay_6   // T56
      := "iJ-magnetTakeDetection3";
   END_TRANSITION
   STEP StoperReset_6:   // S144, max time T#10S, warning time T#7S
              S    "ST10Cylinder".Cy[38].Inout.AutoGoHome
              R    "ST10Cylinder".Cy[38].Inout.AutoGoWork
   END_STEP
   TRANSITION Trans777 FROM StoperReset_6 TO "Process Finish_6"   // T152
      := TRUE;
   END_TRANSITION
   STEP StoperRelease_6:   // S145, max time T#10S, warning time T#7S
              R    "ST10Cylinder".Cy[38].Inout.AutoGoHome
              S    "ST10Cylinder".Cy[38].Inout.AutoGoWork
   END_STEP
   TRANSITION Trans778 FROM StoperRelease_6 TO WaitPalletArrveNextPos_5   // T153
      := #StoperRelease_6.T > t#1000MS;
   END_TRANSITION
   STEP WaitPalletArive_4:   // S146, max time T#10S, warning time T#7S
              N    "AutoProcessControl".Global.J.EmptyStopRequestPallet_2
   END_STEP
   TRANSITION Trans144 FROM WaitPalletArive_4 TO TimeDelay_4   // T155
      := "iJ-magnetTakeDetection2";
   END_TRANSITION
   STEP TimeDelay_4:   // S147, max time T#10S, warning time T#7S
   END_STEP
   TRANSITION Trans146 FROM TimeDelay_4 TO UnloadStoper_2   // T156, jump
      := #TimeDelay_4.T > t#500MS;
   END_TRANSITION
   STEP "CheckMachine Mode_1":   // S154, max time T#10S, warning time T#7S
   END_STEP
   TRANSITION Trans164 FROM "CheckMachine Mode_1" TO LoadingStop_1   // T164
      := NOT "AutoProcessControl".Global.J.EmptyPallet;
   END_TRANSITION
   STEP "Process Finish_7":   // S243, max time T#10S, warning time T#7S
   END_STEP
   TRANSITION Trans256 FROM "Process Finish_7" TO UnloadStoper_3   // T255, jump
      := TRUE;
   END_TRANSITION
   STEP CheckPalletExist_6:   // S57, max time T#10S, warning time T#7S
   END_STEP
   TRANSITION Trans62 FROM CheckPalletExist_6 TO WaitLineMotorReady_6   // T61
      := "iJ-magnetTakeDetection3" AND (#CheckPalletExist_6.T > t#1000MS);
   END_TRANSITION
   TRANSITION Trans148 FROM CheckPalletExist_6 TO WaitPalletArive_5   // T160
      := NOT "iJ-magnetTakeDetection3" AND (#CheckPalletExist_6.T > t#1000MS);
   END_TRANSITION
   STEP AriveTimeDelay_7:   // S148, max time T#10S, warning time T#7S
   END_STEP
   TRANSITION Trans147 FROM AriveTimeDelay_7 TO StoperReset_7   // T157
      := #AriveTimeDelay_7.T > t#500MS;
   END_TRANSITION
   STEP WaitLineMotorReady_6:   // S58, max time T#10S, warning time T#7S
   END_STEP
   TRANSITION Trans63 FROM WaitLineMotorReady_6 TO WaitPalletRequestRelease_6   // T62
      := "MotorControl".Dev[14].OutControl.o_Ready;
   END_TRANSITION
   STEP WaitPalletRequestRelease_6:   // S59, max time T#10S, warning time T#7S
   END_STEP
   TRANSITION Trans64 FROM WaitPalletRequestRelease_6 TO StoperRelease_7   // T63
      := NOT "iJ-magnetTakeShaftDetection";
   END_TRANSITION
   STEP WaitPalletArrveNextPos_6:   // S60, max time T#10S, warning time T#7S
              S    "MotorControl".Dev[14].Auto.Start
              R    "MotorControl".Dev[14].Auto.CCWStart
   END_STEP
   TRANSITION Trans61 FROM WaitPalletArrveNextPos_6 TO AriveTimeDelay_7   // T60
      := "iJ-magnetTakeShaftDetection";
   END_TRANSITION
   STEP StoperReset_7:   // S149, max time T#10S, warning time T#7S
              S    "ST10Cylinder".Cy[39].Inout.AutoGoHome
              R    "ST10Cylinder".Cy[39].Inout.AutoGoWork
   END_STEP
   TRANSITION Trans779 FROM StoperReset_7 TO "Process Finish_7"   // T158
      := TRUE;
   END_TRANSITION
   STEP StoperRelease_7:   // S150, max time T#10S, warning time T#7S
              R    "ST10Cylinder".Cy[39].Inout.AutoGoHome
              S    "ST10Cylinder".Cy[39].Inout.AutoGoWork
   END_STEP
   TRANSITION Trans780 FROM StoperRelease_7 TO WaitPalletArrveNextPos_6   // T159
      := #StoperRelease_7.T > t#1000MS;
   END_TRANSITION
   STEP WaitPalletArive_5:   // S151, max time T#10S, warning time T#7S
              N    "AutoProcessControl".Global.J.EmptyStopRequestPallet_3
   END_STEP
   TRANSITION Trans149 FROM WaitPalletArive_5 TO TimeDelay_5   // T161
      := "iJ-magnetTakeDetection3";
   END_TRANSITION
   STEP TimeDelay_5:   // S152, max time T#10S, warning time T#7S
   END_STEP
   TRANSITION Trans150 FROM TimeDelay_5 TO UnloadStoper_3   // T162, jump
      := #TimeDelay_5.T > t#500MS;
   END_TRANSITION
   STEP "CheckMachine Mode_2":   // S155, max time T#10S, warning time T#7S
   END_STEP
   TRANSITION Trans165 FROM "CheckMachine Mode_2" TO LoadingStop_2   // T165
      := NOT "AutoProcessControl".Global.J.EmptyPallet;
   END_TRANSITION
   STEP "CheckMachine Mode_4":   // S157, max time T#10S, warning time T#7S
   END_STEP
   TRANSITION Trans167 FROM "CheckMachine Mode_4" TO LoadingStop_4   // T167
      := NOT "AutoProcessControl".Global.J.EmptyPallet;
   END_TRANSITION

   // sequencer 3: Empty Process
   INITIAL_STEP CheckMachineMode:   // S200, max time T#10S, warning time T#7S
   END_STEP
   TRANSITION Trans145 FROM CheckMachineMode TO WaitAllStoperReset   // T200
      := "AutoProcessControl".Global.J.EmptyPallet;
   END_TRANSITION
   STEP Step153:   // S153, max time T#10S, warning time T#7S
   END_STEP
   TRANSITION Trans163 FROM Step153 TO "CheckMachine Mode_6"   // T163, jump
      := TRUE;
   END_TRANSITION
   STEP "Process Finish_8":   // S244, max time T#10S, warning time T#7S
   END_STEP
   TRANSITION Trans257 FROM "Process Finish_8" TO Step153   // T256
      := TRUE;
   END_TRANSITION
   STEP LoadStop_14:   // S61, max time T#10S, warning time T#7S
   END_STEP
   TRANSITION Trans154 FROM LoadStop_14 TO CheckPalletExist_10   // T175
      := #LoadStop_14.T > t#2S;
   END_TRANSITION
   STEP LoadStop_12:   // S62, max time T#10S, warning time T#7S
   END_STEP
   TRANSITION Trans152 FROM LoadStop_12 TO CheckPalletExist_8   // T169
      := #LoadStop_12.T > t#2S;
   END_TRANSITION
   STEP "CheckMachine Mode_5":   // S158, max time T#10S, warning time T#7S
   END_STEP
   TRANSITION Trans175 FROM "CheckMachine Mode_5" TO LoadStop_13   // T196
      := "AutoProcessControl".Global.J.EmptyPallet;
   END_TRANSITION
   STEP LoadStop_13:   // S63, max time T#10S, warning time T#7S
   END_STEP
   TRANSITION Trans153 FROM LoadStop_13 TO CheckPalletExist_9   // T170
      := #LoadStop_13.T > t#2S;
   END_TRANSITION
   STEP CheckPalletExist_7:   // S64, max time T#10S, warning time T#7S
   END_STEP
   TRANSITION Trans66 FROM CheckPalletExist_7 TO WaitLineMotorReady_7   // T65
      := "J-mganePalletEmptyCheck1" AND (#CheckPalletExist_7.T > t#1000MS);
   END_TRANSITION
   TRANSITION Trans33 FROM CheckPalletExist_7 TO WaitPalletArive_9   // T32
      := NOT "J-mganePalletEmptyCheck1" AND (#CheckPalletExist_7.T > t#1000MS);
   END_TRANSITION
   STEP AriveTimeDelay_8:   // S159, max time T#10S, warning time T#7S
   END_STEP
   TRANSITION Trans151 FROM AriveTimeDelay_8 TO StoperReset_8   // T168
      := #AriveTimeDelay_8.T > t#500MS;
   END_TRANSITION
   STEP WaitLineMotorReady_7:   // S65, max time T#10S, warning time T#7S
   END_STEP
   TRANSITION Trans67 FROM WaitLineMotorReady_7 TO WaitPalletRequestRelease_7   // T66
      := "MotorControl".Dev[13].OutControl.o_Ready;
   END_TRANSITION
   STEP WaitPalletRequestRelease_7:   // S66, max time T#10S, warning time T#7S
   END_STEP
   TRANSITION Trans68 FROM WaitPalletRequestRelease_7 TO StoperRelease_8   // T67
      := NOT "iJ-magnetTakeGateDetection";
   END_TRANSITION
   STEP LoadStop_11:   // S160, max time T#10S, warning time T#7S
   END_STEP
   TRANSITION Trans781 FROM LoadStop_11 TO CheckPalletExist_7   // T172
      := #LoadStop_11.T > t#2S;
   END_TRANSITION
   STEP WaitPalletArrveNextPos_7:   // S67, max time T#10S, warning time T#7S
   END_STEP
   TRANSITION Trans65 FROM WaitPalletArrveNextPos_7 TO AriveTimeDelay_8   // T64
      := "iJ-magnetTakeGateDetection" OR NOT "AutoProcessControl".Global.J.EmptyPallet;
   END_TRANSITION
   STEP "Process Finish_9":   // S245, max time T#10S, warning time T#7S
   END_STEP
   TRANSITION Trans258 FROM "Process Finish_9" TO "CheckMachine Mode_7"   // T257, jump
      := TRUE;
   END_TRANSITION
   STEP StoperReset_8:   // S161, max time T#10S, warning time T#7S
              S    "ST10Cylinder".Cy[33].Inout.AutoGoHome
              R    "ST10Cylinder".Cy[33].Inout.AutoGoWork
   END_STEP
   TRANSITION Trans782 FROM StoperReset_8 TO "Process Finish_8"   // T173
      := TRUE;
   END_TRANSITION
   STEP StoperRelease_8:   // S162, max time T#10S, warning time T#7S
              R    "ST10Cylinder".Cy[33].Inout.AutoGoHome
              S    "ST10Cylinder".Cy[33].Inout.AutoGoWork
   END_STEP
   TRANSITION Trans783 FROM StoperRelease_8 TO WaitPalletArrveNextPos_7   // T174
      := #StoperRelease_8.T > t#1000MS;
   END_TRANSITION
   STEP CheckPalletExist_8:   // S68, max time T#10S, warning time T#7S
   END_STEP
   TRANSITION Trans70 FROM CheckPalletExist_8 TO WaitLineMotorReady_8   // T69
      := "J-mganePalletEmptyCheck2" AND (#CheckPalletExist_8.T > t#1000MS);
   END_TRANSITION
   TRANSITION Trans156 FROM CheckPalletExist_8 TO WaitPalletArive_6   // T179
      := NOT "J-mganePalletEmptyCheck2" AND (#CheckPalletExist_8.T > t#1000MS);
   END_TRANSITION
   STEP AriveTimeDelay_9:   // S163, max time T#10S, warning time T#7S
   END_STEP
   TRANSITION Trans155 FROM AriveTimeDelay_9 TO StoperReset_9   // T176
      := #AriveTimeDelay_9.T > t#500MS;
   END_TRANSITION
   STEP WaitLineMotorReady_8:   // S69, max time T#10S, warning time T#7S
   END_STEP
   TRANSITION Trans71 FROM WaitLineMotorReady_8 TO WaitPalletRequestRelease_8   // T70
      := "MotorControl".Dev[13].OutControl.o_Ready;
   END_TRANSITION
   STEP WaitPalletRequestRelease_8:   // S70, max time T#10S, warning time T#7S
   END_STEP
   TRANSITION Trans72 FROM WaitPalletRequestRelease_8 TO StoperRelease_9   // T71
      := "AutoProcessControl".Global.J.LoadStopRequestPallet_2;
   END_TRANSITION
   STEP WaitPalletArrveNextPos_8:   // S71, max time T#10S, warning time T#7S
   END_STEP
   TRANSITION Trans69 FROM WaitPalletArrveNextPos_8 TO AriveTimeDelay_9   // T68
      := "J-mganePalletEmptyCheck1";
   END_TRANSITION
   STEP StoperReset_9:   // S164, max time T#10S, warning time T#7S
              S    "ST10Cylinder".Cy[34].Inout.AutoGoHome
              R    "ST10Cylinder".Cy[34].Inout.AutoGoWork
   END_STEP
   TRANSITION Trans784 FROM StoperReset_9 TO "Process Finish_9"   // T177
      := TRUE;
   END_TRANSITION
   STEP StoperRelease_9:   // S165, max time T#10S, warning time T#7S
              R    "ST10Cylinder".Cy[34].Inout.AutoGoHome
              S    "ST10Cylinder".Cy[34].Inout.AutoGoWork
   END_STEP
   TRANSITION Trans785 FROM StoperRelease_9 TO WaitPalletArrveNextPos_8   // T178
      := #StoperRelease_9.T > t#1000MS;
   END_TRANSITION
   STEP WaitPalletArive_6:   // S166, max time T#10S, warning time T#7S
              N    "AutoProcessControl".Global.J.LoadStopRequestPallet_3
   END_STEP
   TRANSITION Trans157 FROM WaitPalletArive_6 TO TimeDelay_6   // T180
      := "J-mganePalletEmptyCheck2" OR NOT "AutoProcessControl".Global.J.EmptyPallet;
   END_TRANSITION
   STEP TimeDelay_6:   // S167, max time T#10S, warning time T#7S
   END_STEP
   TRANSITION Trans158 FROM TimeDelay_6 TO "CheckMachine Mode_7"   // T181, jump
      := #TimeDelay_6.T > t#500MS;
   END_TRANSITION
   STEP "Process Finish_10":   // S246, max time T#10S, warning time T#7S
   END_STEP
   TRANSITION Trans259 FROM "Process Finish_10" TO "CheckMachine Mode_5"   // T258, jump
      := TRUE;
   END_TRANSITION
   STEP CheckPalletExist_9:   // S72, max time T#10S, warning time T#7S
   END_STEP
   TRANSITION Trans74 FROM CheckPalletExist_9 TO WaitLineMotorReady_9   // T73
      := "J-mganePalletEmptyCheck3" AND (#CheckPalletExist_9.T > t#1000MS);
   END_TRANSITION
   TRANSITION Trans160 FROM CheckPalletExist_9 TO WaitPalletArive_7   // T185
      := NOT "J-mganePalletEmptyCheck3" AND (#CheckPalletExist_9.T > t#1000MS);
   END_TRANSITION
   STEP AriveTimeDelay_10:   // S168, max time T#10S, warning time T#7S
   END_STEP
   TRANSITION Trans159 FROM AriveTimeDelay_10 TO StoperReset_10   // T182
      := #AriveTimeDelay_10.T > t#500MS;
   END_TRANSITION
   STEP WaitLineMotorReady_9:   // S73, max time T#10S, warning time T#7S
   END_STEP
   TRANSITION Trans75 FROM WaitLineMotorReady_9 TO WaitPalletRequestRelease_9   // T74
      := "MotorControl".Dev[13].OutControl.o_Ready;
   END_TRANSITION
   STEP WaitPalletRequestRelease_9:   // S74, max time T#10S, warning time T#7S
   END_STEP
   TRANSITION Trans76 FROM WaitPalletRequestRelease_9 TO StoperRelease_10   // T75
      := "AutoProcessControl".Global.J.LoadStopRequestPallet_3;
   END_TRANSITION
   STEP WaitPalletArrveNextPos_9:   // S75, max time T#10S, warning time T#7S
   END_STEP
   TRANSITION Trans73 FROM WaitPalletArrveNextPos_9 TO AriveTimeDelay_10   // T72
      := "J-mganePalletEmptyCheck2";
   END_TRANSITION
   STEP StoperReset_10:   // S169, max time T#10S, warning time T#7S
              S    "ST10Cylinder".Cy[35].Inout.AutoGoHome
              R    "ST10Cylinder".Cy[35].Inout.AutoGoWork
   END_STEP
   TRANSITION Trans786 FROM StoperReset_10 TO "Process Finish_10"   // T183
      := TRUE;
   END_TRANSITION
   STEP StoperRelease_10:   // S170, max time T#10S, warning time T#7S
              R    "ST10Cylinder".Cy[35].Inout.AutoGoHome
              S    "ST10Cylinder".Cy[35].Inout.AutoGoWork
   END_STEP
   TRANSITION Trans787 FROM StoperRelease_10 TO WaitPalletArrveNextPos_9   // T184
      := #StoperRelease_10.T > t#1000MS;
   END_TRANSITION
   STEP WaitPalletArive_7:   // S171, max time T#10S, warning time T#7S
              N    "AutoProcessControl".Global.J.LoadStopRequestPallet_4
   END_STEP
   TRANSITION Trans161 FROM WaitPalletArive_7 TO TimeDelay_7   // T186
      := "J-mganePalletEmptyCheck3" OR NOT "AutoProcessControl".Global.J.EmptyPallet;
   END_TRANSITION
   STEP TimeDelay_7:   // S172, max time T#10S, warning time T#7S
   END_STEP
   TRANSITION Trans162 FROM TimeDelay_7 TO "CheckMachine Mode_5"   // T187, jump
      := #TimeDelay_7.T > t#500MS;
   END_TRANSITION
   STEP "Process Finish_11":   // S247, max time T#10S, warning time T#7S
   END_STEP
   TRANSITION Trans260 FROM "Process Finish_11" TO "CheckMachine Mode_8"   // T259, jump
      := TRUE;
   END_TRANSITION
   STEP CheckPalletExist_10:   // S76, max time T#10S, warning time T#7S
   END_STEP
   TRANSITION Trans78 FROM CheckPalletExist_10 TO WaitLineMotorReady_10   // T77
      := "J-mganePalletEmptyCheck4" AND "iJ-MagnetMiddleDetection" AND (#CheckPalletExist_10.T > t#1000MS);
   END_TRANSITION
   TRANSITION Trans170 FROM CheckPalletExist_10 TO WaitPalletArive_8   // T191
      := NOT "J-mganePalletEmptyCheck4" AND (#CheckPalletExist_10.T > t#1000MS);
   END_TRANSITION
   STEP AriveTimeDelay_11:   // S173, max time T#10S, warning time T#7S
   END_STEP
   TRANSITION Trans169 FROM AriveTimeDelay_11 TO StoperReset_11   // T188
      := #AriveTimeDelay_11.T > t#500MS;
   END_TRANSITION
   STEP WaitLineMotorReady_10:   // S77, max time T#10S, warning time T#7S
   END_STEP
   TRANSITION Trans79 FROM WaitLineMotorReady_10 TO WaitPalletRequestRelease_10   // T78
      := "MotorControl".Dev[13].OutControl.o_Ready;
   END_TRANSITION
   STEP WaitPalletRequestRelease_10:   // S78, max time T#10S, warning time T#7S
   END_STEP
   TRANSITION Trans80 FROM WaitPalletRequestRelease_10 TO StoperRelease_11   // T79
      := "AutoProcessControl".Global.J.LoadStopRequestPallet_4;
   END_TRANSITION
   STEP WaitPalletArrveNextPos_10:   // S79, max time T#10S, warning time T#7S
   END_STEP
   TRANSITION Trans77 FROM WaitPalletArrveNextPos_10 TO AriveTimeDelay_11   // T76
      := "J-mganePalletEmptyCheck3";
   END_TRANSITION
   STEP StoperReset_11:   // S174, max time T#10S, warning time T#7S
              S    "ST10Cylinder".Cy[36].Inout.AutoGoHome
              R    "ST10Cylinder".Cy[36].Inout.AutoGoWork
   END_STEP
   TRANSITION Trans788 FROM StoperReset_11 TO "Process Finish_11"   // T189
      := TRUE;
   END_TRANSITION
   STEP StoperRelease_11:   // S175, max time T#10S, warning time T#7S
              R    "ST10Cylinder".Cy[36].Inout.AutoGoHome
              S    "ST10Cylinder".Cy[36].Inout.AutoGoWork
   END_STEP
   TRANSITION Trans789 FROM StoperRelease_11 TO WaitPalletArrveNextPos_10   // T190
      := #StoperRelease_11.T > t#1000MS;
   END_TRANSITION
   STEP WaitPalletArive_8:   // S176, max time T#10S, warning time T#7S
   END_STEP
   TRANSITION Trans171 FROM WaitPalletArive_8 TO TimeDelay_8   // T192
      := ("J-mganePalletEmptyCheck4" AND "iJ-MagnetMiddleDetection") OR NOT "AutoProcessControl".Global.J.EmptyPallet;
   END_TRANSITION
   STEP TimeDelay_8:   // S177, max time T#10S, warning time T#7S
   END_STEP
   TRANSITION Trans172 FROM TimeDelay_8 TO "CheckMachine Mode_8"   // T193, jump
      := #TimeDelay_8.T > t#500MS;
   END_TRANSITION
   STEP "CheckMachine Mode_6":   // S178, max time T#10S, warning time T#7S
   END_STEP
   TRANSITION Trans173 FROM "CheckMachine Mode_6" TO LoadStop_11   // T194
      := "AutoProcessControl".Global.J.EmptyPallet;
   END_TRANSITION
   STEP "CheckMachine Mode_7":   // S179, max time T#10S, warning time T#7S
   END_STEP
   TRANSITION Trans174 FROM "CheckMachine Mode_7" TO LoadStop_12   // T195
      := "AutoProcessControl".Global.J.EmptyPallet;
   END_TRANSITION
   STEP "CheckMachine Mode_8":   // S180, max time T#10S, warning time T#7S
   END_STEP
   TRANSITION Trans168 FROM "CheckMachine Mode_8" TO LoadStop_14   // T171
      := "AutoProcessControl".Global.J.EmptyPallet;
   END_TRANSITION
   STEP WaitAllStoperReset:   // S181, max time T#10S, warning time T#7S
   END_STEP
   TRANSITION Trans197 FROM WaitAllStoperReset TO MotorRun_1   // T197
      := "ST10Cylinder".Cy[33].Inout.AutoGoHome AND NOT "ST10Cylinder".Cy[33].Inout.AutoGoWork AND "ST10Cylinder".Cy[34].Inout.AutoGoHome AND NOT "ST10Cylinder".Cy[34].Inout.AutoGoWork AND "ST10Cylinder".Cy[35].Inout.AutoGoHome AND NOT "ST10Cylinder".Cy[35].Inout.AutoGoWork AND "ST10Cylinder".Cy[36].Inout.AutoGoHome AND NOT "ST10Cylinder".Cy[36].Inout.AutoGoWork;
   END_TRANSITION
   STEP Step182:   // S182, max time T#10S, warning time T#7S
   END_STEP
   TRANSITION Trans198 FROM Step182 TO ("CheckMachine Mode_7", "CheckMachine Mode_5", "CheckMachine Mode_8", "CheckMachine Mode_6")   // T198
      := TRUE;
   END_TRANSITION
   STEP MotorRun_1:   // S80, max time T#10S, warning time T#7S
              R    "MotorControl".Dev[13].Auto.Start
              S    "MotorControl".Dev[13].Auto.CCWStart
              S    "MotorControl".Dev[14].Auto.Start
              R    "MotorControl".Dev[14].Auto.CCWStart
   END_STEP
   TRANSITION Trans81 FROM MotorRun_1 TO Step182   // T80
      := TRUE;
   END_TRANSITION
   STEP WaitPalletArive_9:   // S183, max time T#10S, warning time T#7S
              N    "AutoProcessControl".Global.J.LoadStopRequestPallet_2
   END_STEP
   TRANSITION Trans176 FROM WaitPalletArive_9 TO TimeDelay_9   // T199
      := "J-mganePalletEmptyCheck1" OR NOT "AutoProcessControl".Global.J.EmptyPallet;
   END_TRANSITION
   STEP TimeDelay_9:   // S184, max time T#10S, warning time T#7S
   END_STEP
   TRANSITION Trans177 FROM TimeDelay_9 TO "CheckMachine Mode_6"   // T201, jump
      := #TimeDelay_9.T > t#500MS;
   END_TRANSITION

   // permanent post-instructions
   NETWORK 1
      #ioPM_Inface.StepNum := #RT_DATA.S_DISPLAY;
   NETWORK 2
      IF #iSysInface.Reset THEN #AlarmID := 0; END_IF;
   NETWORK 3
      #TON[10].TON(IN := #工件放行中, PT := T#0.5S);
      IF #TON[10].Q THEN #工件放行中 := FALSE; END_IF;
END_FUNCTION_BLOCK

FUNCTION_BLOCK "ST10_Flow27_KReserveLoad&Unload"   // FB1097, GRAPH
// stored: AcknowledgeErrorsRequired false, AutoNumber false, GraphVersion 6.0, InitialValuesAcquisition false, SetENOAutomatically false
   // inherited from GRAPH_BASE
   VAR_INPUT
      iSysInface : "RCS_SysComInterface_V1";
   END_VAR
   VAR_IN_OUT
      ioPM_Inface : "RCS_PMInterface_V1";
      ioStatus : Int;
   END_VAR
   VAR
      sCtrlMode { S7_SetPoint := 'True'} : "SysFlowCtrlGraph";
      sUpdMES_Data : Bool;   // 更新MES数据
      工件放行中 : Bool;
      前站站号 { ExternalAccessible := 'False'; ExternalVisible := 'False'; ExternalWritable := 'False'} : UInt;
      本站站号 { ExternalAccessible := 'False'; ExternalVisible := 'False'; ExternalWritable := 'False'} : UInt;
      弹窗Temp : Array[1..10] of Int;
      AlarmID : Int;
      TON { S7_SetPoint := 'True'} : Array[0..10] of TON_TIME;
      TOF { S7_SetPoint := 'True'} : Array[0..10] of TOF_TIME;
      sUP { S7_SetPoint := 'True'} : Array[0..10] of Bool;
      更新RFID完成 : Bool;
   END_VAR
   VAR_TEMP
      Tempresult : USInt;
      本站站号乘10 : UInt;
   END_VAR
   // // TON[0] : 托盘流入1托盘到位传感器 / iA-Rotating product Check
   // // TON[1] : 托盘流入1托盘到位传感器
   // // TON[2] : 托盘流入1产品有无传感器
   // // TON[3] : 托盘流入1产品有无传感器
   // // TON[4] : 托盘流入1姿态检测光电2
   // // TON[5] : 托盘流入1姿态检测光电3
   // // TON[0].Q : 托盘流入1托盘到位 / iA-Rotating product Check
   // // TON[1].Q : 托盘流入1托盘无
   // // TON[2].Q : 托盘流入1有产品
   // // TON[3].Q : 托盘流入1无产品
   // // TON[4].Q : 托盘流入1姿态检测光电2
   // // TON[5].Q : 托盘流入1姿态检测光电3
   // // TOF[1] : iA-Rotating product Check
BEGIN
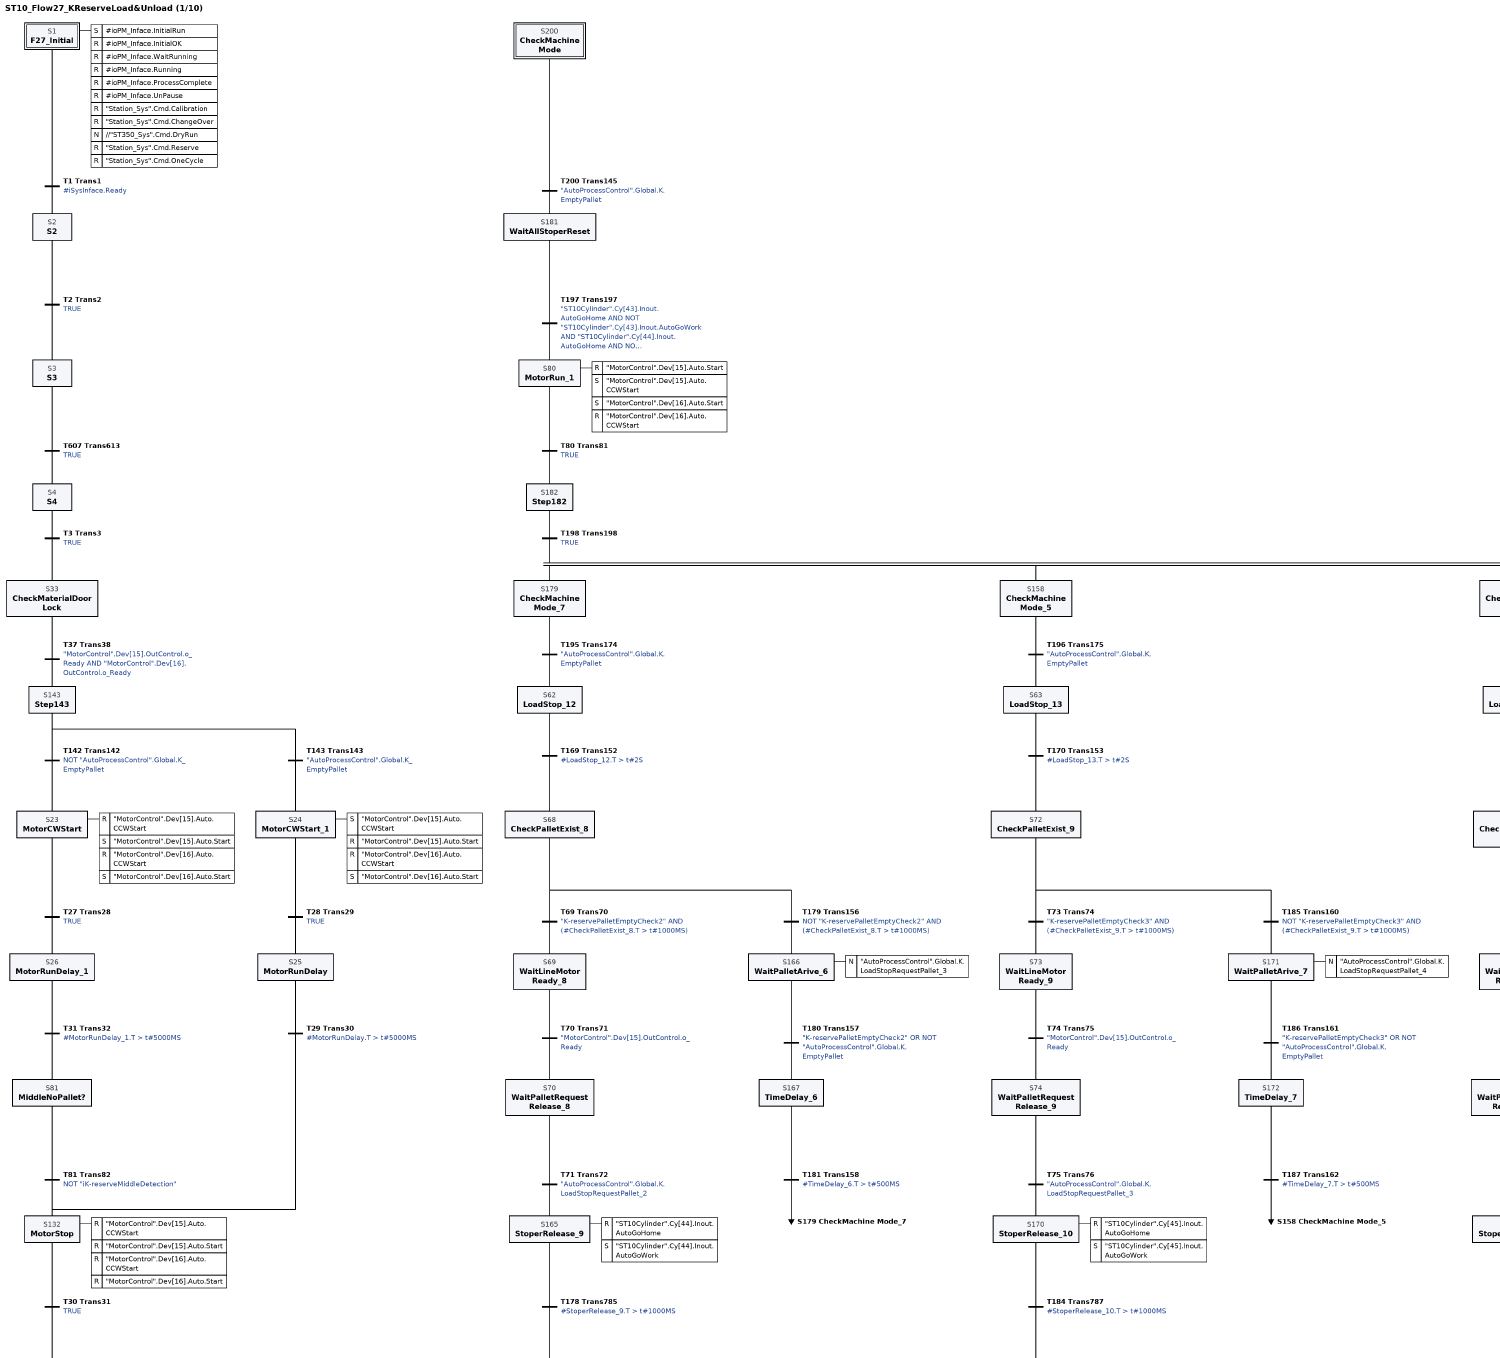
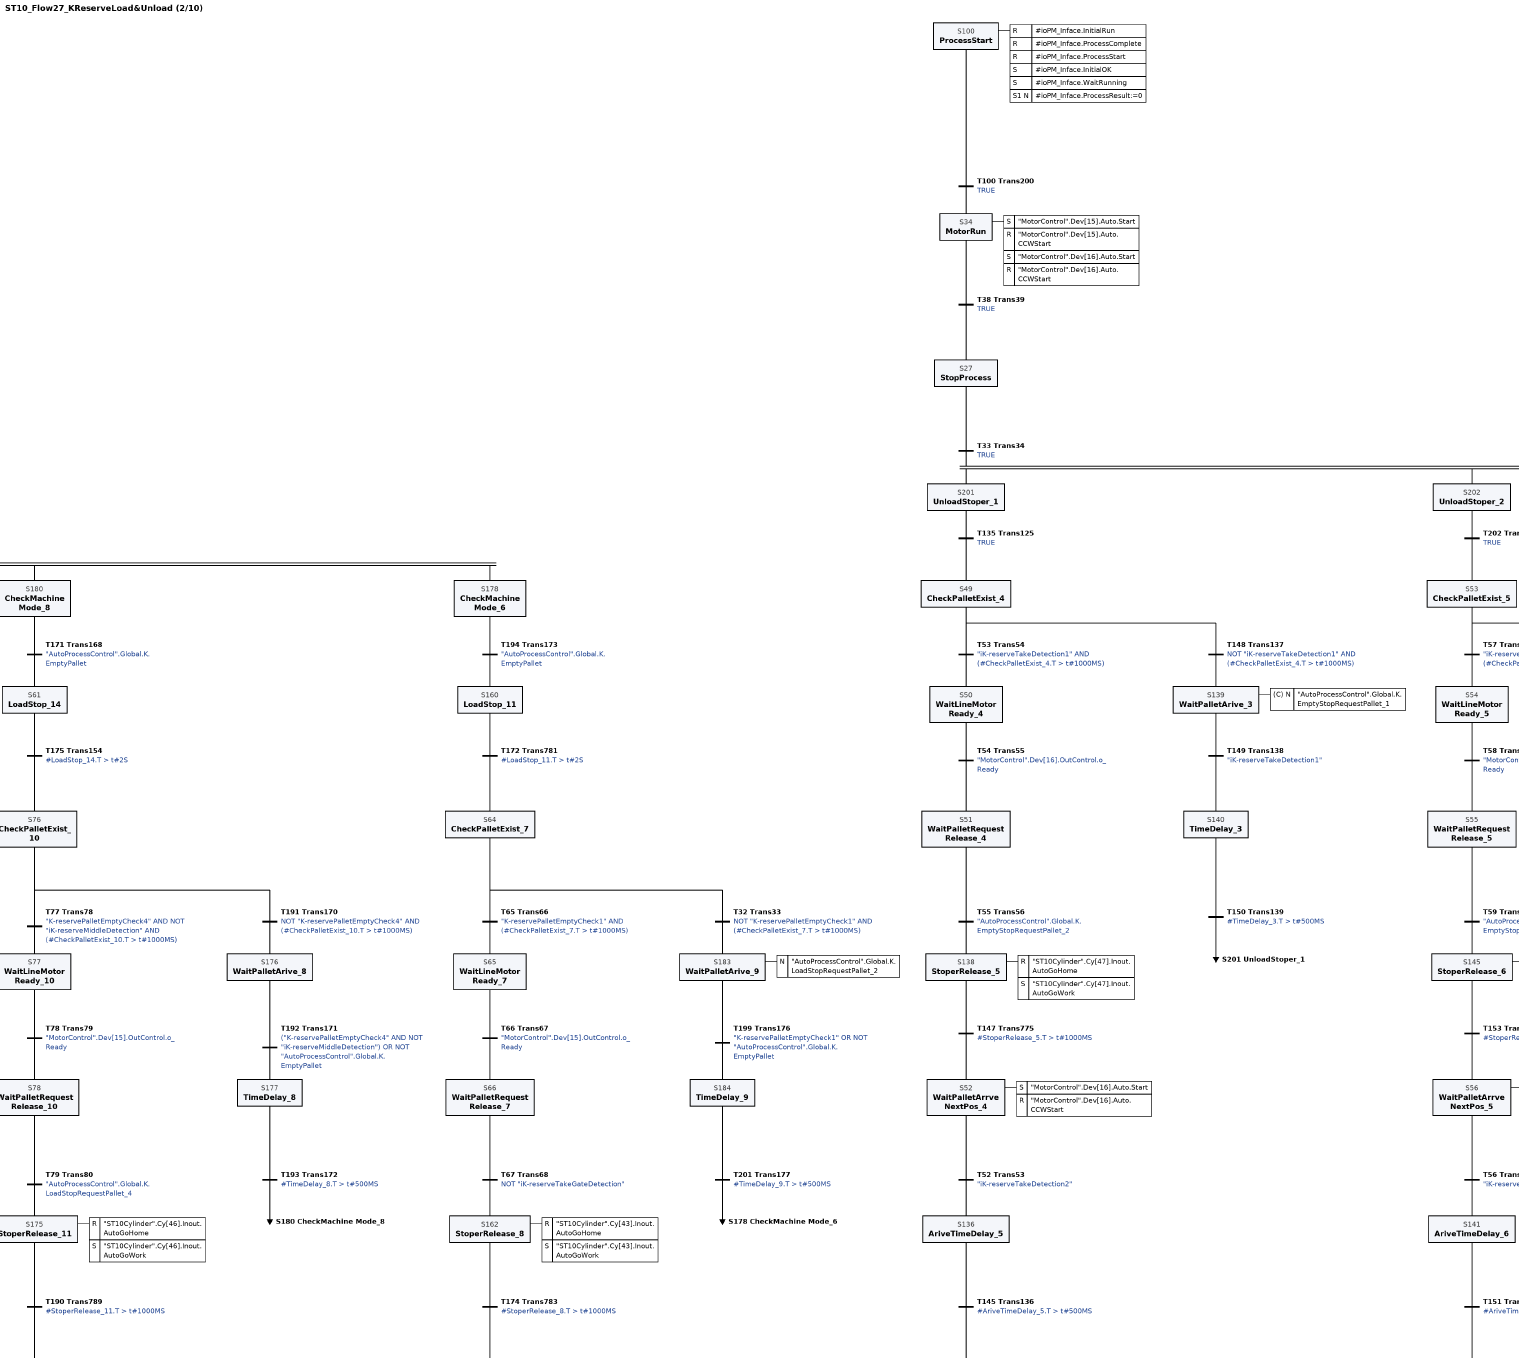
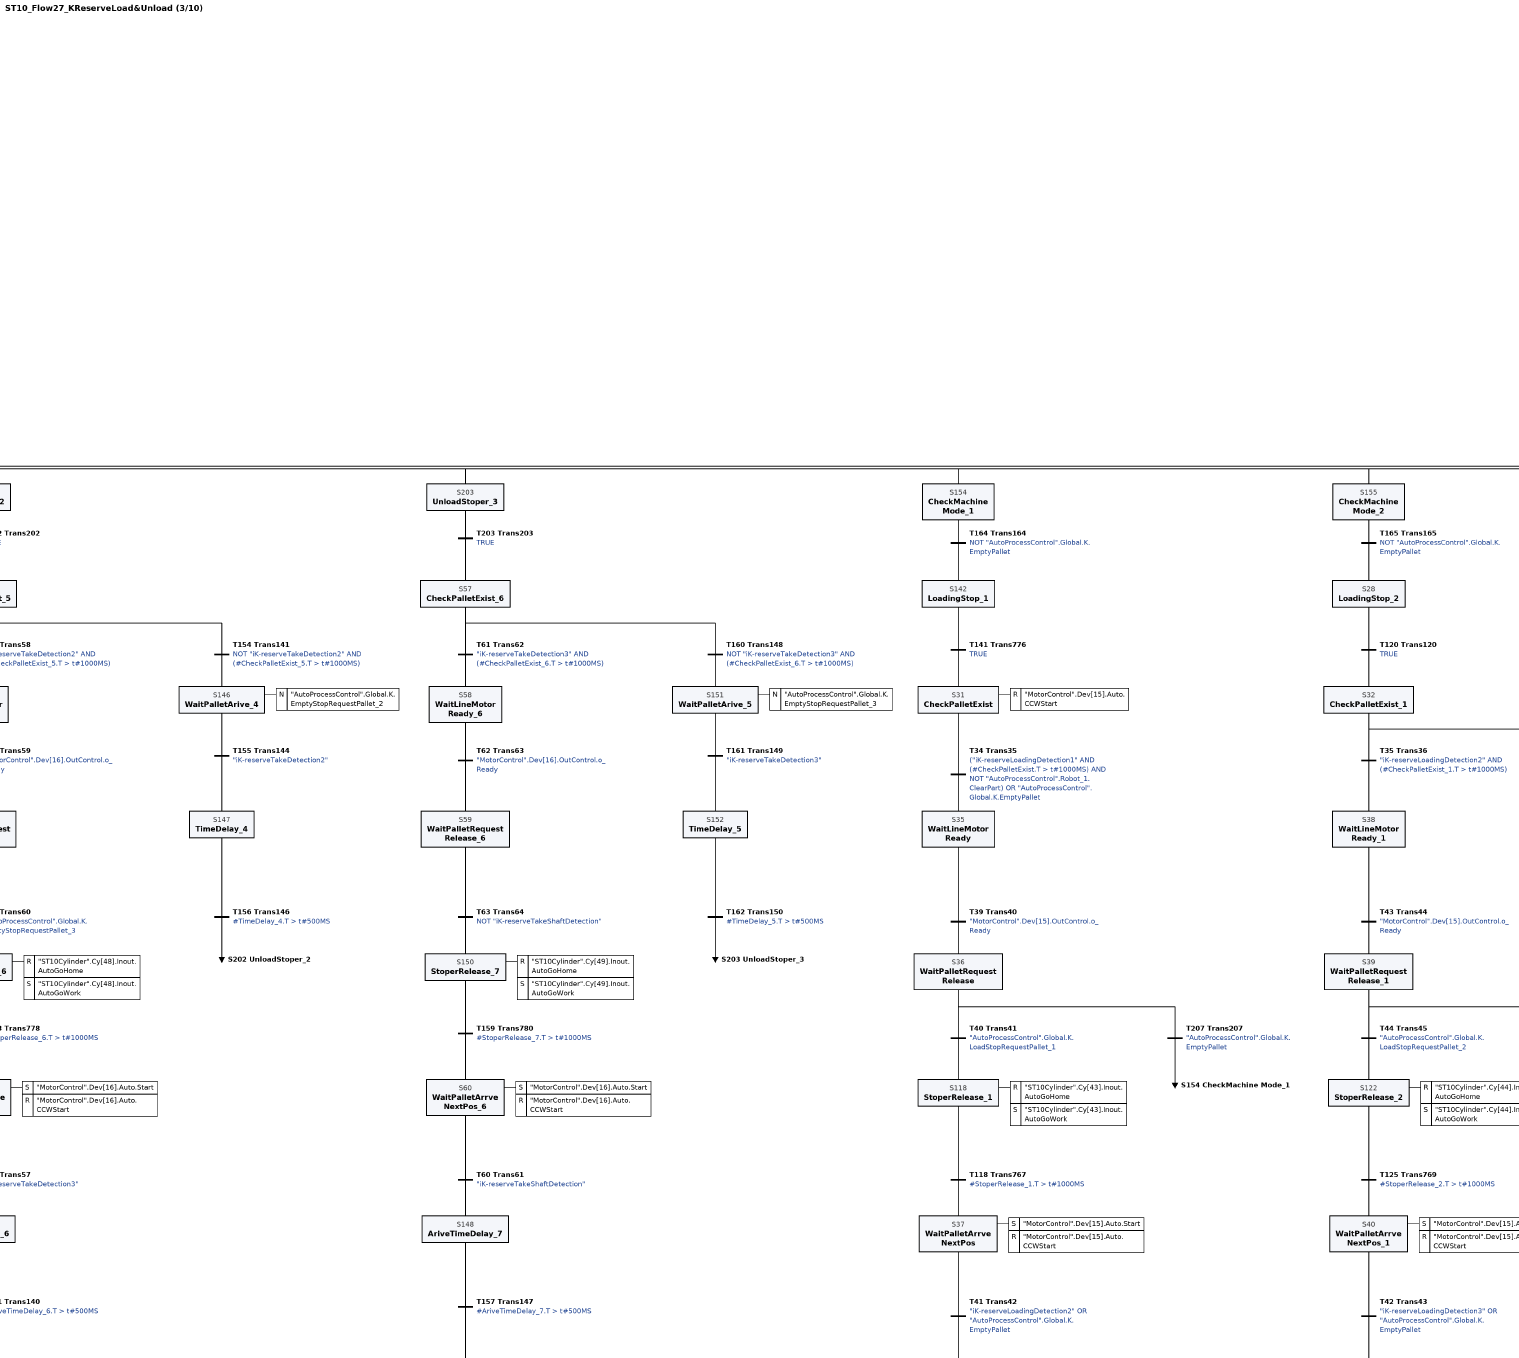
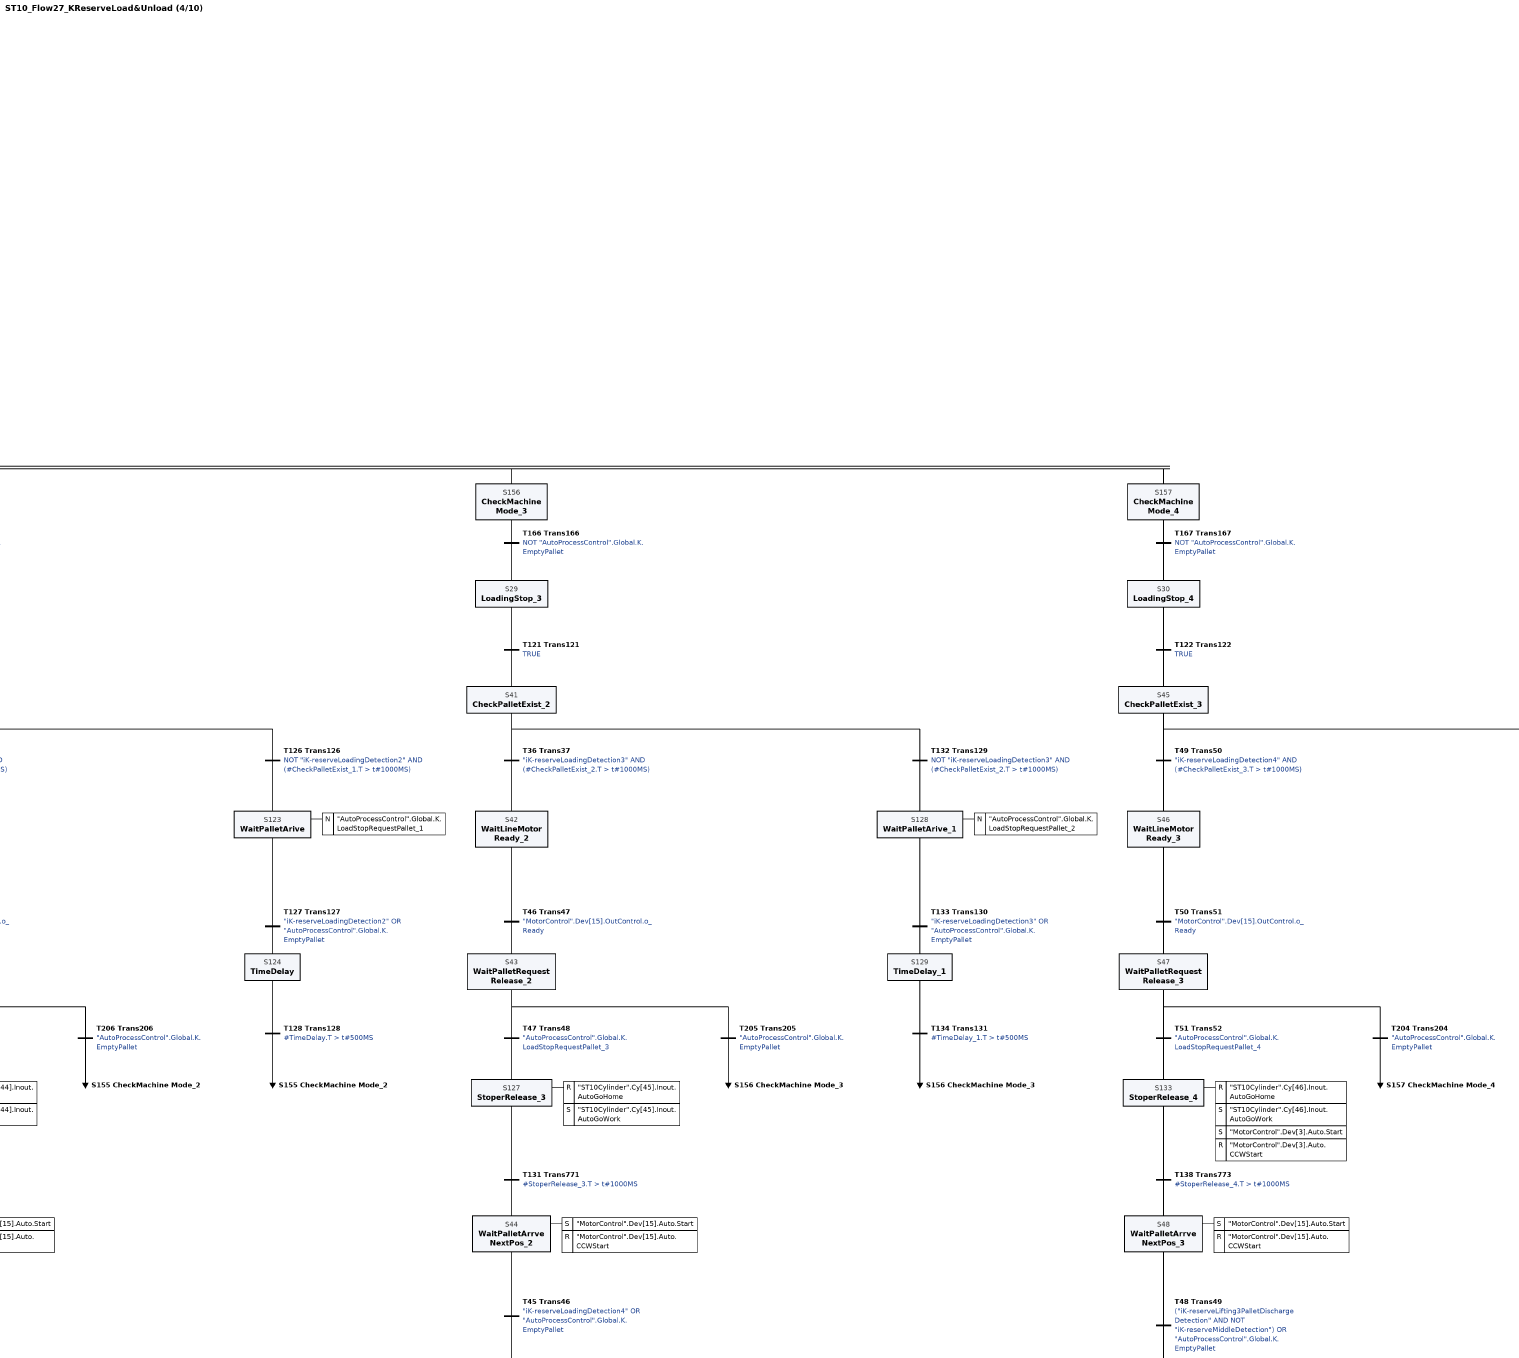
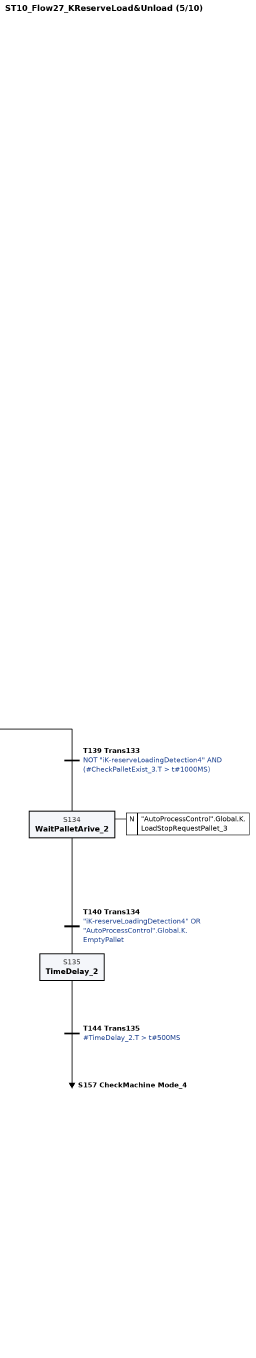
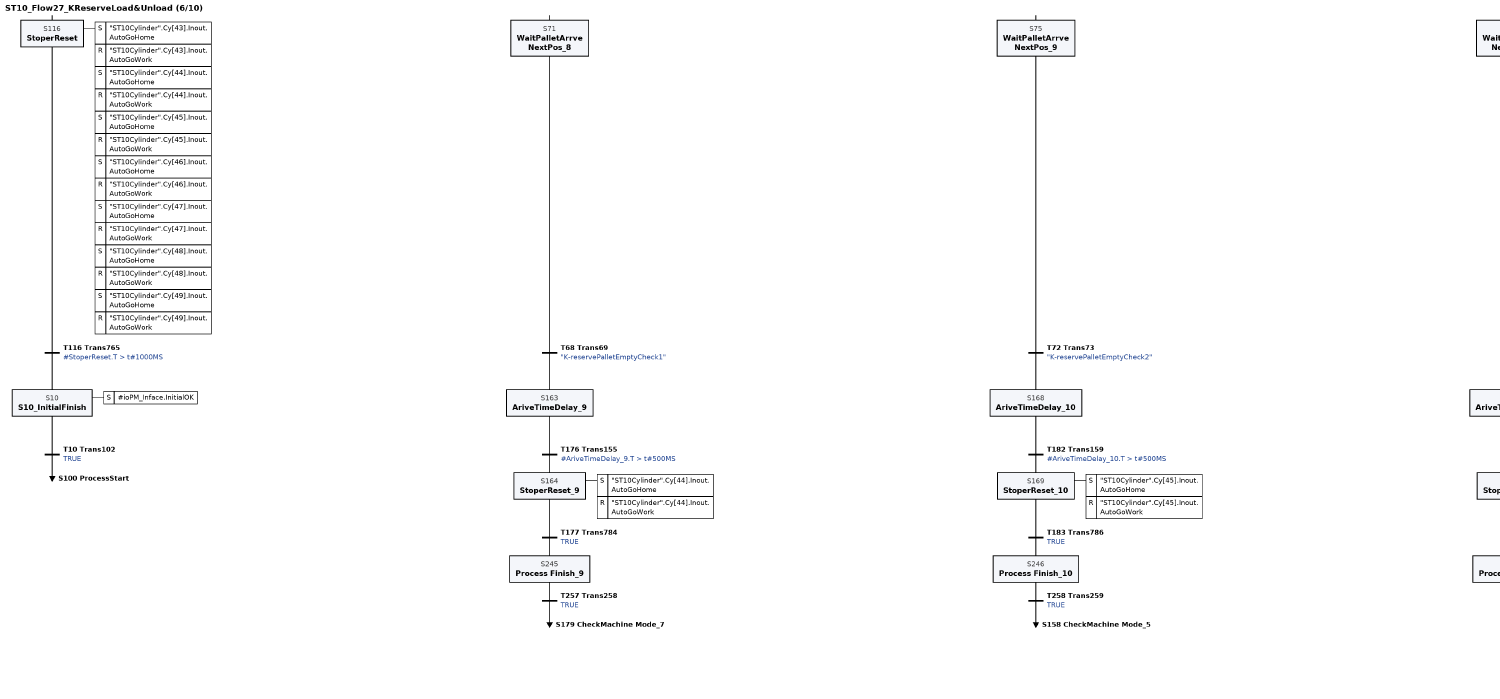
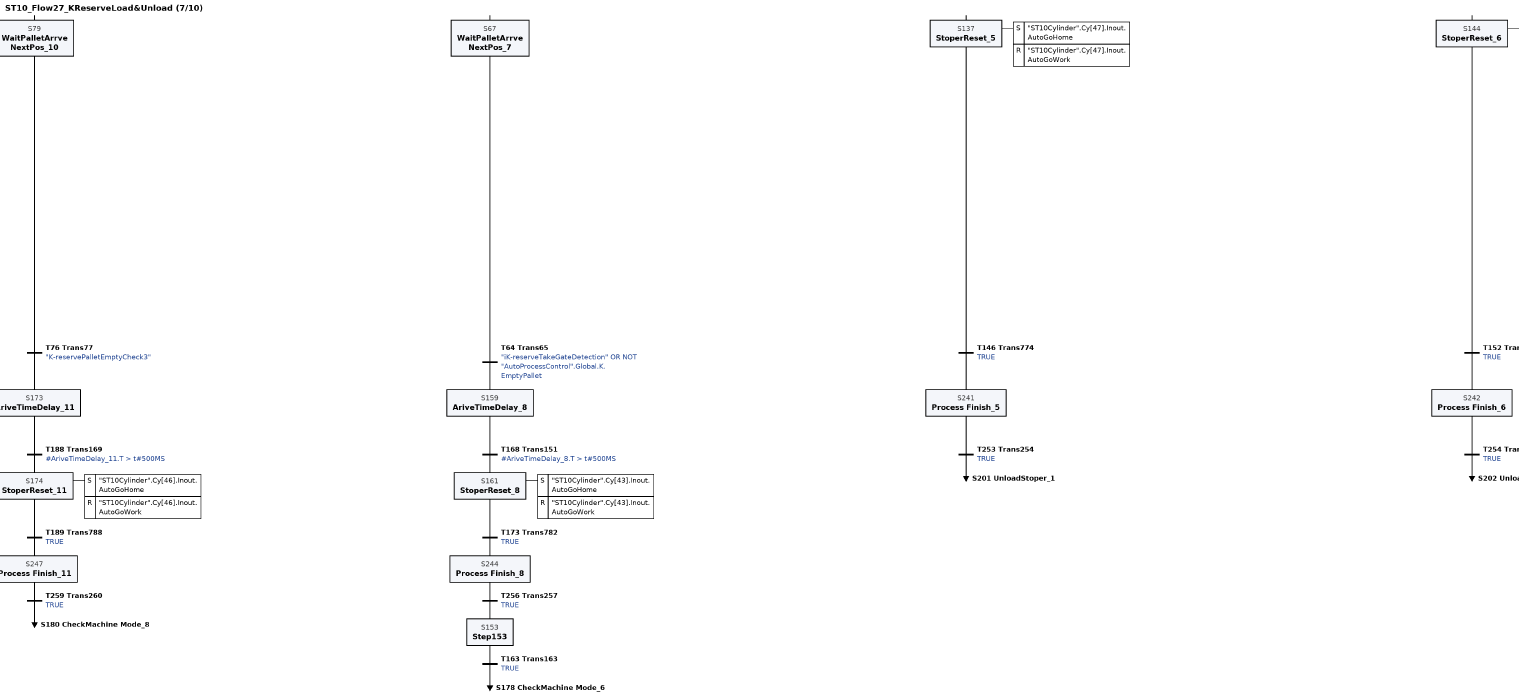
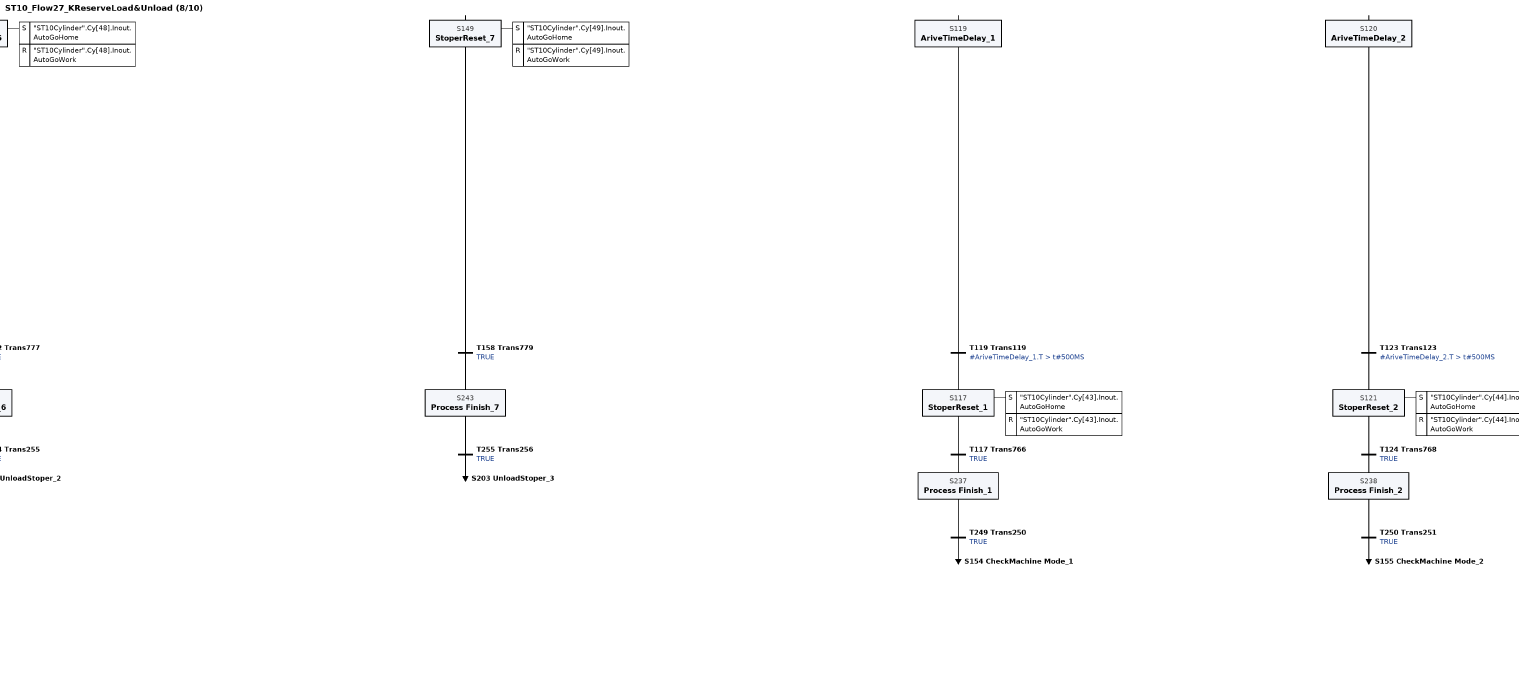
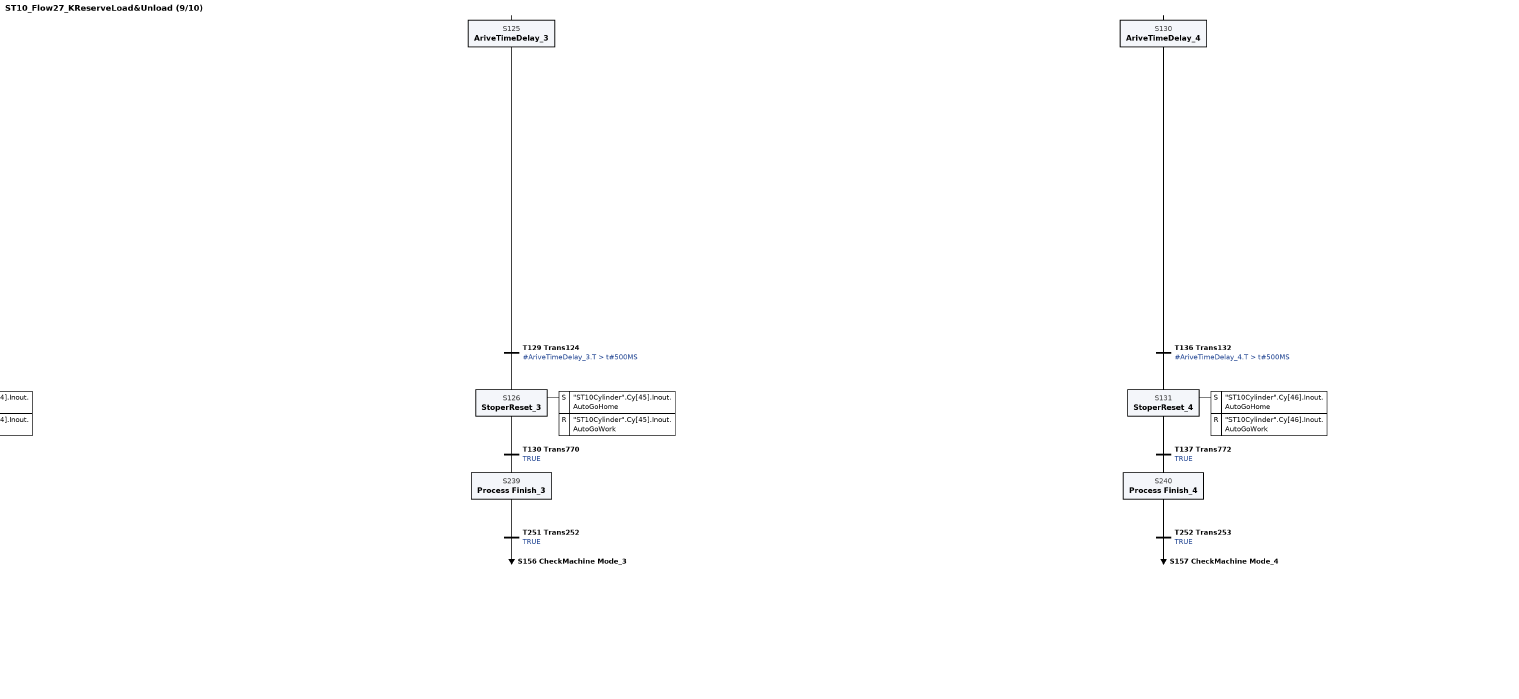
   // permanent pre-instructions
   NETWORK 1
      #TON[10].TON(IN := "AlwaysTRUE" AND "Station_Sys".Alarm.ImmediatelyStop, PT := T#300ms);
      #ioPM_Inface.AlarmImdilyStop := #TON[10].Q;
      #ioPM_Inface.AlarmCycleStop := "AlwaysTRUE" AND "Station_Sys".Alarm.CycleStop;
   NETWORK 2
      IF NOT False THEN
          #sCtrlMode(iSysInface := #iSysInface, ioPM_Inface := #ioPM_Inface, ioGraphCtrl := #RT_DATA.MOP);   // "SysFlowCtrlGraph"
      END_IF;
   NETWORK 3
      #TON[0].TON(IN := "AlwaysTRUE" AND "iK-reserveLifting3PalletDischargeDetection", PT := t#2000ms);   // 工位11有托盘
      #TOF[1].TOF(IN := "AlwaysTRUE" AND NOT "iK-reserveLifting3PalletDischargeDetection", PT := T#300ms);   // 工位无托盘
      #TON[2].TON(IN := "AlwaysTRUE", PT := T#300ms);
      #TOF[3].TOF(IN := "AlwaysTRUE", PT := T#300ms);
      #TON[4].TON(IN := "AlwaysTRUE", PT := T#300ms);
      #TOF[5].TOF(IN := "AlwaysTRUE", PT := T#300ms);
   NETWORK 4
      #前站站号 := 345;
      #本站站号 := 350;

   // sequencer 1: S01-S99 初始化 / S01-S99 Initial
   INITIAL_STEP F27_Initial:   // S1, max time T#10S, warning time T#7S
              S    #ioPM_Inface.InitialRun
              R    #ioPM_Inface.InitialOK
              R    #ioPM_Inface.WaitRunning
              R    #ioPM_Inface.Running
              R    #ioPM_Inface.ProcessComplete
              R    #ioPM_Inface.UnPause
              R    "Station_Sys".Cmd.Calibration
              R    "Station_Sys".Cmd.ChangeOver
                   //"ST350_Sys".Cmd.DryRun
              R    "Station_Sys".Cmd.Reserve
              R    "Station_Sys".Cmd.OneCycle
   END_STEP
   TRANSITION Trans1 FROM F27_Initial TO S2   // T1
      := #iSysInface.Ready;
   END_TRANSITION
   STEP S2:   // S2, max time T#10S, warning time T#7S
   END_STEP
   TRANSITION Trans2 FROM S2 TO S3   // T2
      := TRUE;
   END_TRANSITION
   STEP S4:   // S4, max time T#10S, warning time T#7S
   END_STEP
   TRANSITION Trans3 FROM S4 TO CheckMaterialDoorLock   // T3
      := TRUE;
   END_TRANSITION
   STEP MotorRunDelay_1:   // S26, max time T#10S, warning time T#7S
   END_STEP
   TRANSITION Trans32 FROM MotorRunDelay_1 TO "MiddleNoPallet?"   // T31
      := #MotorRunDelay_1.T > t#5000MS;
   END_TRANSITION
   STEP S10_InitialFinish:   // S10, max time T#10S, warning time T#7S
              S    #ioPM_Inface.InitialOK
   END_STEP
   TRANSITION Trans102 FROM S10_InitialFinish TO ProcessStart   // T10, jump
      := TRUE;
   END_TRANSITION
   STEP S3:   // S3, max time T#10S, warning time T#7S
   END_STEP
   TRANSITION Trans613 FROM S3 TO S4   // T607
      := TRUE;
   END_TRANSITION
   STEP CheckMaterialDoorLock:   // S33, max time T#10S, warning time T#7S
   END_STEP
   TRANSITION Trans38 FROM CheckMaterialDoorLock TO Step143   // T37
      := "MotorControl".Dev[15].OutControl.o_Ready AND "MotorControl".Dev[16].OutControl.o_Ready;
   END_TRANSITION
   STEP "MiddleNoPallet?":   // S81, max time T#10S, warning time T#7S
   END_STEP
   TRANSITION Trans82 FROM "MiddleNoPallet?" TO MotorStop   // T81
      := NOT "iK-reserveMiddleDetection";
   END_TRANSITION
   STEP StoperReset:   // S116, max time T#10S, warning time T#7S
              S    "ST10Cylinder".Cy[43].Inout.AutoGoHome
              R    "ST10Cylinder".Cy[43].Inout.AutoGoWork
              S    "ST10Cylinder".Cy[44].Inout.AutoGoHome
              R    "ST10Cylinder".Cy[44].Inout.AutoGoWork
              S    "ST10Cylinder".Cy[45].Inout.AutoGoHome
              R    "ST10Cylinder".Cy[45].Inout.AutoGoWork
              S    "ST10Cylinder".Cy[46].Inout.AutoGoHome
              R    "ST10Cylinder".Cy[46].Inout.AutoGoWork
              S    "ST10Cylinder".Cy[47].Inout.AutoGoHome
              R    "ST10Cylinder".Cy[47].Inout.AutoGoWork
              S    "ST10Cylinder".Cy[48].Inout.AutoGoHome
              R    "ST10Cylinder".Cy[48].Inout.AutoGoWork
              S    "ST10Cylinder".Cy[49].Inout.AutoGoHome
              R    "ST10Cylinder".Cy[49].Inout.AutoGoWork
   END_STEP
   TRANSITION Trans765 FROM StoperReset TO S10_InitialFinish   // T116
      := #StoperReset.T > t#1000MS;
   END_TRANSITION
   STEP MotorCWStart_1:   // S24, max time T#10S, warning time T#7S
              S    "MotorControl".Dev[15].Auto.CCWStart
              R    "MotorControl".Dev[15].Auto.Start
              R    "MotorControl".Dev[16].Auto.CCWStart
              S    "MotorControl".Dev[16].Auto.Start
   END_STEP
   TRANSITION Trans29 FROM MotorCWStart_1 TO MotorRunDelay   // T28
      := TRUE;
   END_TRANSITION
   STEP Step143:   // S143, max time T#10S, warning time T#7S
   END_STEP
   TRANSITION Trans142 FROM Step143 TO MotorCWStart   // T142
      := NOT "AutoProcessControl".Global.K_EmptyPallet;
   END_TRANSITION
   TRANSITION Trans143 FROM Step143 TO MotorCWStart_1   // T143
      := "AutoProcessControl".Global.K_EmptyPallet;
   END_TRANSITION
   STEP MotorCWStart:   // S23, max time T#10S, warning time T#7S
              R    "MotorControl".Dev[15].Auto.CCWStart
              S    "MotorControl".Dev[15].Auto.Start
              R    "MotorControl".Dev[16].Auto.CCWStart
              S    "MotorControl".Dev[16].Auto.Start
   END_STEP
   TRANSITION Trans28 FROM MotorCWStart TO MotorRunDelay_1   // T27
      := TRUE;
   END_TRANSITION
   STEP MotorStop:   // S132, max time T#10S, warning time T#7S
              R    "MotorControl".Dev[15].Auto.CCWStart
              R    "MotorControl".Dev[15].Auto.Start
              R    "MotorControl".Dev[16].Auto.CCWStart
              R    "MotorControl".Dev[16].Auto.Start
   END_STEP
   TRANSITION Trans31 FROM MotorStop TO StoperReset   // T30
      := TRUE;
   END_TRANSITION
   STEP MotorRunDelay:   // S25, max time T#10S, warning time T#7S
   END_STEP
   TRANSITION Trans30 FROM MotorRunDelay TO MotorStop   // T29
      := #MotorRunDelay.T > t#5000MS;
   END_TRANSITION

